    !***********************************************************
    !
    ! Procedure main
    !
    !   This is the entry point of your program
    !
    !***********************************************************
    PROC main()
        Path_10;
      !Add your code here
    ENDPROC
      PROC Path_10()
SetDO drillDone,0;
MoveAbsJ jHome, v100, fine, tool0\WObj:= wobj0;
WaitTime 2;
confL \Off;
confJ \Off;
        MoveJ RelTool(Target_10,0,0,-10),v60,z10,DrillTool\WObj:=FakeWing;
SetDO drillDone,1;
WaitUntil drillDone = 0;
        MoveL Target_10,v30,fine,DrillTool\WObj:=FakeWing;
SetDO drillDone,1;
WaitUntil drillDone = 0;
        MoveL RelTool(Target_10,0,0,-10),v30,z10,DrillTool\WObj:=FakeWing;
        MoveL RelTool(Target_20,0,0,-10),v30,z10,DrillTool\WObj:=FakeWing;
        MoveL Target_20,v30,fine,DrillTool\WObj:=FakeWing;
SetDO drillDone,1;
WaitUntil drillDone = 0;
        MoveL RelTool(Target_20,0,0,-10),v30,z10,DrillTool\WObj:=FakeWing;
        MoveL RelTool(Target_30,0,0,-10),v30,z10,DrillTool\WObj:=FakeWing;
        MoveL Target_30,v30,fine,DrillTool\WObj:=FakeWing;
SetDO drillDone,1;
WaitUntil drillDone = 0;
        MoveL RelTool(Target_30,0,0,-10),v30,z10,DrillTool\WObj:=FakeWing;
        MoveL RelTool(Target_40,0,0,-10),v30,z10,DrillTool\WObj:=FakeWing;
        MoveL Target_40,v30,fine,DrillTool\WObj:=FakeWing;
SetDO drillDone,1;
WaitUntil drillDone = 0;
        MoveL RelTool(Target_40,0,0,-10),v30,z10,DrillTool\WObj:=FakeWing;
        MoveL RelTool(Target_50,0,0,-10),v30,z10,DrillTool\WObj:=FakeWing;
        MoveL Target_50,v30,fine,DrillTool\WObj:=FakeWing;
SetDO drillDone,1;
WaitUntil drillDone = 0;
        MoveL RelTool(Target_50,0,0,-10),v30,z10,DrillTool\WObj:=FakeWing;
        MoveL RelTool(Target_60,0,0,-10),v30,z10,DrillTool\WObj:=FakeWing;
        MoveL Target_60,v30,fine,DrillTool\WObj:=FakeWing;
SetDO drillDone,1;
WaitUntil drillDone = 0;
        MoveL RelTool(Target_60,0,0,-10),v30,z10,DrillTool\WObj:=FakeWing;
        MoveL RelTool(Target_70,0,0,-10),v30,z10,DrillTool\WObj:=FakeWing;
        MoveL Target_70,v30,fine,DrillTool\WObj:=FakeWing;
SetDO drillDone,1;
WaitUntil drillDone = 0;
        MoveL RelTool(Target_70,0,0,-10),v30,z10,DrillTool\WObj:=FakeWing;
        MoveL RelTool(Target_80,0,0,-10),v30,z10,DrillTool\WObj:=FakeWing;
        MoveL Target_80,v30,fine,DrillTool\WObj:=FakeWing;
SetDO drillDone,1;
WaitUntil drillDone = 0;
        MoveL RelTool(Target_80,0,0,-10),v30,z10,DrillTool\WObj:=FakeWing;
        MoveL RelTool(Target_90,0,0,-10),v30,z10,DrillTool\WObj:=FakeWing;
        MoveL Target_90,v30,fine,DrillTool\WObj:=FakeWing;
SetDO drillDone,1;
WaitUntil drillDone = 0;
        MoveL RelTool(Target_90,0,0,-10),v30,z10,DrillTool\WObj:=FakeWing;
        MoveL RelTool(Target_100,0,0,-10),v30,z10,DrillTool\WObj:=FakeWing;
        MoveL Target_100,v30,fine,DrillTool\WObj:=FakeWing;
SetDO drillDone,1;
WaitUntil drillDone = 0;
        MoveL RelTool(Target_100,0,0,-10),v30,z10,DrillTool\WObj:=FakeWing;
        MoveL RelTool(Target_110,0,0,-10),v30,z10,DrillTool\WObj:=FakeWing;
        MoveL Target_110,v30,fine,DrillTool\WObj:=FakeWing;
SetDO drillDone,1;
WaitUntil drillDone = 0;
        MoveL RelTool(Target_110,0,0,-10),v30,z10,DrillTool\WObj:=FakeWing;
        MoveL RelTool(Target_120,0,0,-10),v30,z10,DrillTool\WObj:=FakeWing;
        MoveL Target_120,v30,fine,DrillTool\WObj:=FakeWing;
SetDO drillDone,1;
WaitUntil drillDone = 0;
        MoveL RelTool(Target_120,0,0,-10),v30,z10,DrillTool\WObj:=FakeWing;
        MoveL RelTool(Target_130,0,0,-10),v30,z10,DrillTool\WObj:=FakeWing;
        MoveL Target_130,v30,fine,DrillTool\WObj:=FakeWing;
SetDO drillDone,1;
WaitUntil drillDone = 0;
        MoveL RelTool(Target_130,0,0,-10),v30,z10,DrillTool\WObj:=FakeWing;
        MoveL RelTool(Target_140,0,0,-10),v30,z10,DrillTool\WObj:=FakeWing;
        MoveL Target_140,v30,fine,DrillTool\WObj:=FakeWing;
SetDO drillDone,1;
WaitUntil drillDone = 0;
        MoveL RelTool(Target_140,0,0,-10),v30,z10,DrillTool\WObj:=FakeWing;
        MoveL RelTool(Target_150,0,0,-10),v30,z10,DrillTool\WObj:=FakeWing;
        MoveL Target_150,v30,fine,DrillTool\WObj:=FakeWing;
SetDO drillDone,1;
WaitUntil drillDone = 0;
        MoveL RelTool(Target_150,0,0,-10),v30,z10,DrillTool\WObj:=FakeWing;
        MoveL RelTool(Target_160,0,0,-10),v30,z10,DrillTool\WObj:=FakeWing;
        MoveL Target_160,v30,fine,DrillTool\WObj:=FakeWing;
SetDO drillDone,1;
WaitUntil drillDone = 0;
        MoveL RelTool(Target_160,0,0,-10),v30,z10,DrillTool\WObj:=FakeWing;
        MoveL RelTool(Target_170,0,0,-10),v30,z10,DrillTool\WObj:=FakeWing;
        MoveL Target_170,v30,fine,DrillTool\WObj:=FakeWing;
SetDO drillDone,1;
WaitUntil drillDone = 0;
        MoveL RelTool(Target_170,0,0,-10),v30,z10,DrillTool\WObj:=FakeWing;
        MoveL RelTool(Target_180,0,0,-10),v30,z10,DrillTool\WObj:=FakeWing;
        MoveL Target_180,v30,fine,DrillTool\WObj:=FakeWing;
SetDO drillDone,1;
WaitUntil drillDone = 0;
        MoveL RelTool(Target_180,0,0,-10),v30,z10,DrillTool\WObj:=FakeWing;
        MoveL RelTool(Target_190,0,0,-10),v30,z10,DrillTool\WObj:=FakeWing;
        MoveL Target_190,v30,fine,DrillTool\WObj:=FakeWing;
SetDO drillDone,1;
WaitUntil drillDone = 0;
        MoveL RelTool(Target_190,0,0,-10),v30,z10,DrillTool\WObj:=FakeWing;
        MoveL RelTool(Target_200,0,0,-10),v30,z10,DrillTool\WObj:=FakeWing;
        MoveL Target_200,v30,fine,DrillTool\WObj:=FakeWing;
SetDO drillDone,1;
WaitUntil drillDone = 0;
        MoveL RelTool(Target_200,0,0,-10),v30,z10,DrillTool\WObj:=FakeWing;
        MoveL RelTool(Target_210,0,0,-10),v30,z10,DrillTool\WObj:=FakeWing;
        MoveL Target_210,v30,fine,DrillTool\WObj:=FakeWing;
SetDO drillDone,1;
WaitUntil drillDone = 0;
        MoveL RelTool(Target_210,0,0,-10),v30,z10,DrillTool\WObj:=FakeWing;
        MoveL RelTool(Target_220,0,0,-10),v30,z10,DrillTool\WObj:=FakeWing;
        MoveL Target_220,v30,fine,DrillTool\WObj:=FakeWing;
SetDO drillDone,1;
WaitUntil drillDone = 0;
        MoveL RelTool(Target_220,0,0,-10),v30,z10,DrillTool\WObj:=FakeWing;
        MoveL RelTool(Target_230,0,0,-10),v30,z10,DrillTool\WObj:=FakeWing;
        MoveL Target_230,v30,fine,DrillTool\WObj:=FakeWing;
SetDO drillDone,1;
WaitUntil drillDone = 0;
        MoveL RelTool(Target_230,0,0,-10),v30,z10,DrillTool\WObj:=FakeWing;
        MoveL RelTool(Target_240,0,0,-10),v30,z10,DrillTool\WObj:=FakeWing;
        MoveL Target_240,v30,fine,DrillTool\WObj:=FakeWing;
SetDO drillDone,1;
WaitUntil drillDone = 0;
        MoveL RelTool(Target_240,0,0,-10),v30,z10,DrillTool\WObj:=FakeWing;
        MoveL RelTool(Target_250,0,0,-10),v30,z10,DrillTool\WObj:=FakeWing;
        MoveL Target_250,v30,fine,DrillTool\WObj:=FakeWing;
SetDO drillDone,1;
WaitUntil drillDone = 0;
        MoveL RelTool(Target_250,0,0,-10),v30,z10,DrillTool\WObj:=FakeWing;
        MoveL RelTool(Target_260,0,0,-10),v30,z10,DrillTool\WObj:=FakeWing;
        MoveL Target_260,v30,fine,DrillTool\WObj:=FakeWing;
SetDO drillDone,1;
WaitUntil drillDone = 0;
        MoveL RelTool(Target_260,0,0,-10),v30,z10,DrillTool\WObj:=FakeWing;
        MoveL RelTool(Target_270,0,0,-10),v30,z10,DrillTool\WObj:=FakeWing;
        MoveL Target_270,v30,fine,DrillTool\WObj:=FakeWing;
SetDO drillDone,1;
WaitUntil drillDone = 0;
        MoveL RelTool(Target_270,0,0,-10),v30,z10,DrillTool\WObj:=FakeWing;
        MoveL RelTool(Target_280,0,0,-10),v30,z10,DrillTool\WObj:=FakeWing;
        MoveL Target_280,v30,fine,DrillTool\WObj:=FakeWing;
SetDO drillDone,1;
WaitUntil drillDone = 0;
        MoveL RelTool(Target_280,0,0,-10),v30,z10,DrillTool\WObj:=FakeWing;
        MoveL RelTool(Target_290,0,0,-10),v30,z10,DrillTool\WObj:=FakeWing;
        MoveL Target_290,v30,fine,DrillTool\WObj:=FakeWing;
SetDO drillDone,1;
WaitUntil drillDone = 0;
        MoveL RelTool(Target_290,0,0,-10),v30,z10,DrillTool\WObj:=FakeWing;
        MoveL RelTool(Target_300,0,0,-10),v30,z10,DrillTool\WObj:=FakeWing;
        MoveL Target_300,v30,fine,DrillTool\WObj:=FakeWing;
SetDO drillDone,1;
WaitUntil drillDone = 0;
        MoveL RelTool(Target_300,0,0,-10),v30,z10,DrillTool\WObj:=FakeWing;
        MoveL RelTool(Target_310,0,0,-10),v30,z10,DrillTool\WObj:=FakeWing;
        MoveL Target_310,v30,fine,DrillTool\WObj:=FakeWing;
SetDO drillDone,1;
WaitUntil drillDone = 0;
        MoveL RelTool(Target_310,0,0,-10),v30,z10,DrillTool\WObj:=FakeWing;
        MoveL RelTool(Target_320,0,0,-10),v30,z10,DrillTool\WObj:=FakeWing;
        MoveL Target_320,v30,fine,DrillTool\WObj:=FakeWing;
SetDO drillDone,1;
WaitUntil drillDone = 0;
        MoveL RelTool(Target_320,0,0,-10),v30,z10,DrillTool\WObj:=FakeWing;
        MoveL RelTool(Target_330,0,0,-10),v30,z10,DrillTool\WObj:=FakeWing;
        MoveL Target_330,v30,fine,DrillTool\WObj:=FakeWing;
SetDO drillDone,1;
WaitUntil drillDone = 0;
        MoveL RelTool(Target_330,0,0,-10),v30,z10,DrillTool\WObj:=FakeWing;
        MoveL RelTool(Target_340,0,0,-10),v30,z10,DrillTool\WObj:=FakeWing;
        MoveL Target_340,v30,fine,DrillTool\WObj:=FakeWing;
SetDO drillDone,1;
WaitUntil drillDone = 0;
        MoveL RelTool(Target_340,0,0,-10),v30,z10,DrillTool\WObj:=FakeWing;
        MoveL RelTool(Target_350,0,0,-10),v30,z10,DrillTool\WObj:=FakeWing;
        MoveL Target_350,v30,fine,DrillTool\WObj:=FakeWing;
SetDO drillDone,1;
WaitUntil drillDone = 0;
        MoveL RelTool(Target_350,0,0,-10),v30,z10,DrillTool\WObj:=FakeWing;
        MoveL RelTool(Target_360,0,0,-10),v30,z10,DrillTool\WObj:=FakeWing;
        MoveL Target_360,v30,fine,DrillTool\WObj:=FakeWing;
SetDO drillDone,1;
WaitUntil drillDone = 0;
        MoveL RelTool(Target_360,0,0,-10),v30,z10,DrillTool\WObj:=FakeWing;
        MoveL RelTool(Target_370,0,0,-10),v30,z10,DrillTool\WObj:=FakeWing;
        MoveL Target_370,v30,fine,DrillTool\WObj:=FakeWing;
SetDO drillDone,1;
WaitUntil drillDone = 0;
        MoveL RelTool(Target_370,0,0,-10),v30,z10,DrillTool\WObj:=FakeWing;
        MoveL RelTool(Target_380,0,0,-10),v30,z10,DrillTool\WObj:=FakeWing;
        MoveL Target_380,v30,fine,DrillTool\WObj:=FakeWing;
SetDO drillDone,1;
WaitUntil drillDone = 0;
        MoveL RelTool(Target_380,0,0,-10),v30,z10,DrillTool\WObj:=FakeWing;
        MoveL RelTool(Target_390,0,0,-10),v30,z10,DrillTool\WObj:=FakeWing;
        MoveL Target_390,v30,fine,DrillTool\WObj:=FakeWing;
SetDO drillDone,1;
WaitUntil drillDone = 0;
        MoveL RelTool(Target_390,0,0,-10),v30,z10,DrillTool\WObj:=FakeWing;
        MoveL RelTool(Target_400,0,0,-10),v30,z10,DrillTool\WObj:=FakeWing;
        MoveL Target_400,v30,fine,DrillTool\WObj:=FakeWing;
SetDO drillDone,1;
WaitUntil drillDone = 0;
        MoveL RelTool(Target_400,0,0,-10),v30,z10,DrillTool\WObj:=FakeWing;
        MoveL RelTool(Target_410,0,0,-10),v30,z10,DrillTool\WObj:=FakeWing;
        MoveL Target_410,v30,fine,DrillTool\WObj:=FakeWing;
SetDO drillDone,1;
WaitUntil drillDone = 0;
        MoveL RelTool(Target_410,0,0,-10),v30,z10,DrillTool\WObj:=FakeWing;
        MoveL RelTool(Target_420,0,0,-10),v30,z10,DrillTool\WObj:=FakeWing;
        MoveL Target_420,v30,fine,DrillTool\WObj:=FakeWing;
SetDO drillDone,1;
WaitUntil drillDone = 0;
        MoveL RelTool(Target_420,0,0,-10),v30,z10,DrillTool\WObj:=FakeWing;
        MoveL RelTool(Target_430,0,0,-10),v30,z10,DrillTool\WObj:=FakeWing;
        MoveL Target_430,v30,fine,DrillTool\WObj:=FakeWing;
SetDO drillDone,1;
WaitUntil drillDone = 0;
        MoveL RelTool(Target_430,0,0,-10),v30,z10,DrillTool\WObj:=FakeWing;
        MoveL RelTool(Target_440,0,0,-10),v30,z10,DrillTool\WObj:=FakeWing;
        MoveL Target_440,v30,fine,DrillTool\WObj:=FakeWing;
SetDO drillDone,1;
WaitUntil drillDone = 0;
        MoveL RelTool(Target_440,0,0,-10),v30,z10,DrillTool\WObj:=FakeWing;
        MoveL RelTool(Target_450,0,0,-10),v30,z10,DrillTool\WObj:=FakeWing;
        MoveL Target_450,v30,fine,DrillTool\WObj:=FakeWing;
SetDO drillDone,1;
WaitUntil drillDone = 0;
        MoveL RelTool(Target_450,0,0,-10),v30,z10,DrillTool\WObj:=FakeWing;
        MoveL RelTool(Target_460,0,0,-10),v30,z10,DrillTool\WObj:=FakeWing;
        MoveL Target_460,v30,fine,DrillTool\WObj:=FakeWing;
SetDO drillDone,1;
WaitUntil drillDone = 0;
        MoveL RelTool(Target_460,0,0,-10),v30,z10,DrillTool\WObj:=FakeWing;
        MoveL RelTool(Target_470,0,0,-10),v30,z10,DrillTool\WObj:=FakeWing;
        MoveL Target_470,v30,fine,DrillTool\WObj:=FakeWing;
SetDO drillDone,1;
WaitUntil drillDone = 0;
        MoveL RelTool(Target_470,0,0,-10),v30,z10,DrillTool\WObj:=FakeWing;
        MoveL RelTool(Target_480,0,0,-10),v30,z10,DrillTool\WObj:=FakeWing;
        MoveL Target_480,v30,fine,DrillTool\WObj:=FakeWing;
SetDO drillDone,1;
WaitUntil drillDone = 0;
        MoveL RelTool(Target_480,0,0,-10),v30,z10,DrillTool\WObj:=FakeWing;
        MoveL RelTool(Target_490,0,0,-10),v30,z10,DrillTool\WObj:=FakeWing;
        MoveL Target_490,v30,fine,DrillTool\WObj:=FakeWing;
SetDO drillDone,1;
WaitUntil drillDone = 0;
        MoveL RelTool(Target_490,0,0,-10),v30,z10,DrillTool\WObj:=FakeWing;
        MoveL RelTool(Target_500,0,0,-10),v30,z10,DrillTool\WObj:=FakeWing;
        MoveL Target_500,v30,fine,DrillTool\WObj:=FakeWing;
SetDO drillDone,1;
WaitUntil drillDone = 0;
        MoveL RelTool(Target_500,0,0,-10),v30,z10,DrillTool\WObj:=FakeWing;
        MoveL RelTool(Target_510,0,0,-10),v30,z10,DrillTool\WObj:=FakeWing;
        MoveL Target_510,v30,fine,DrillTool\WObj:=FakeWing;
SetDO drillDone,1;
WaitUntil drillDone = 0;
        MoveL RelTool(Target_510,0,0,-10),v30,z10,DrillTool\WObj:=FakeWing;
        MoveL RelTool(Target_520,0,0,-10),v30,z10,DrillTool\WObj:=FakeWing;
        MoveL Target_520,v30,fine,DrillTool\WObj:=FakeWing;
SetDO drillDone,1;
WaitUntil drillDone = 0;
        MoveL RelTool(Target_520,0,0,-10),v30,z10,DrillTool\WObj:=FakeWing;
        MoveL RelTool(Target_530,0,0,-10),v30,z10,DrillTool\WObj:=FakeWing;
        MoveL Target_530,v30,fine,DrillTool\WObj:=FakeWing;
SetDO drillDone,1;
WaitUntil drillDone = 0;
        MoveL RelTool(Target_530,0,0,-10),v30,z10,DrillTool\WObj:=FakeWing;
        MoveL RelTool(Target_540,0,0,-10),v30,z10,DrillTool\WObj:=FakeWing;
        MoveL Target_540,v30,fine,DrillTool\WObj:=FakeWing;
SetDO drillDone,1;
WaitUntil drillDone = 0;
        MoveL RelTool(Target_540,0,0,-10),v30,z10,DrillTool\WObj:=FakeWing;
        MoveL RelTool(Target_550,0,0,-10),v30,z10,DrillTool\WObj:=FakeWing;
        MoveL Target_550,v30,fine,DrillTool\WObj:=FakeWing;
SetDO drillDone,1;
WaitUntil drillDone = 0;
        MoveL RelTool(Target_550,0,0,-10),v30,z10,DrillTool\WObj:=FakeWing;
        MoveL RelTool(Target_560,0,0,-10),v30,z10,DrillTool\WObj:=FakeWing;
        MoveL Target_560,v30,fine,DrillTool\WObj:=FakeWing;
SetDO drillDone,1;
WaitUntil drillDone = 0;
        MoveL RelTool(Target_560,0,0,-10),v30,z10,DrillTool\WObj:=FakeWing;
        MoveL RelTool(Target_570,0,0,-10),v30,z10,DrillTool\WObj:=FakeWing;
        MoveL Target_570,v30,fine,DrillTool\WObj:=FakeWing;
SetDO drillDone,1;
WaitUntil drillDone = 0;
        MoveL RelTool(Target_570,0,0,-10),v30,z10,DrillTool\WObj:=FakeWing;
        MoveL RelTool(Target_580,0,0,-10),v30,z10,DrillTool\WObj:=FakeWing;
        MoveL Target_580,v30,fine,DrillTool\WObj:=FakeWing;
SetDO drillDone,1;
WaitUntil drillDone = 0;
        MoveL RelTool(Target_580,0,0,-10),v30,z10,DrillTool\WObj:=FakeWing;
        MoveL RelTool(Target_590,0,0,-10),v30,z10,DrillTool\WObj:=FakeWing;
        MoveL Target_590,v30,fine,DrillTool\WObj:=FakeWing;
SetDO drillDone,1;
WaitUntil drillDone = 0;
        MoveL RelTool(Target_590,0,0,-10),v30,z10,DrillTool\WObj:=FakeWing;
        MoveL RelTool(Target_600,0,0,-10),v30,z10,DrillTool\WObj:=FakeWing;
        MoveL Target_600,v30,fine,DrillTool\WObj:=FakeWing;
SetDO drillDone,1;
WaitUntil drillDone = 0;
        MoveL RelTool(Target_600,0,0,-10),v30,z10,DrillTool\WObj:=FakeWing;
        MoveL RelTool(Target_610,0,0,-10),v30,z10,DrillTool\WObj:=FakeWing;
        MoveL Target_610,v30,fine,DrillTool\WObj:=FakeWing;
SetDO drillDone,1;
WaitUntil drillDone = 0;
        MoveL RelTool(Target_610,0,0,-10),v30,z10,DrillTool\WObj:=FakeWing;
        MoveL RelTool(Target_620,0,0,-10),v30,z10,DrillTool\WObj:=FakeWing;
        MoveL Target_620,v30,fine,DrillTool\WObj:=FakeWing;
SetDO drillDone,1;
WaitUntil drillDone = 0;
        MoveL RelTool(Target_620,0,0,-10),v30,z10,DrillTool\WObj:=FakeWing;
        MoveL RelTool(Target_630,0,0,-10),v30,z10,DrillTool\WObj:=FakeWing;
        MoveL Target_630,v30,fine,DrillTool\WObj:=FakeWing;
SetDO drillDone,1;
WaitUntil drillDone = 0;
        MoveL RelTool(Target_630,0,0,-10),v30,z10,DrillTool\WObj:=FakeWing;
        MoveL RelTool(Target_640,0,0,-10),v30,z10,DrillTool\WObj:=FakeWing;
        MoveL Target_640,v30,fine,DrillTool\WObj:=FakeWing;
SetDO drillDone,1;
WaitUntil drillDone = 0;
        MoveL RelTool(Target_640,0,0,-10),v30,z10,DrillTool\WObj:=FakeWing;
        MoveL RelTool(Target_650,0,0,-10),v30,z10,DrillTool\WObj:=FakeWing;
        MoveL Target_650,v30,fine,DrillTool\WObj:=FakeWing;
SetDO drillDone,1;
WaitUntil drillDone = 0;
        MoveL RelTool(Target_650,0,0,-10),v30,z10,DrillTool\WObj:=FakeWing;
        MoveL RelTool(Target_660,0,0,-10),v30,z10,DrillTool\WObj:=FakeWing;
        MoveL Target_660,v30,fine,DrillTool\WObj:=FakeWing;
SetDO drillDone,1;
WaitUntil drillDone = 0;
        MoveL RelTool(Target_660,0,0,-10),v30,z10,DrillTool\WObj:=FakeWing;
        MoveL RelTool(Target_670,0,0,-10),v30,z10,DrillTool\WObj:=FakeWing;
        MoveL Target_670,v30,fine,DrillTool\WObj:=FakeWing;
SetDO drillDone,1;
WaitUntil drillDone = 0;
        MoveL RelTool(Target_670,0,0,-10),v30,z10,DrillTool\WObj:=FakeWing;
        MoveL RelTool(Target_680,0,0,-10),v30,z10,DrillTool\WObj:=FakeWing;
        MoveL Target_680,v30,fine,DrillTool\WObj:=FakeWing;
SetDO drillDone,1;
WaitUntil drillDone = 0;
        MoveL RelTool(Target_680,0,0,-10),v30,z10,DrillTool\WObj:=FakeWing;
        MoveL RelTool(Target_690,0,0,-10),v30,z10,DrillTool\WObj:=FakeWing;
        MoveL Target_690,v30,fine,DrillTool\WObj:=FakeWing;
SetDO drillDone,1;
WaitUntil drillDone = 0;
        MoveL RelTool(Target_690,0,0,-10),v30,z10,DrillTool\WObj:=FakeWing;
        MoveL RelTool(Target_700,0,0,-10),v30,z10,DrillTool\WObj:=FakeWing;
        MoveL Target_700,v30,fine,DrillTool\WObj:=FakeWing;
SetDO drillDone,1;
WaitUntil drillDone = 0;
        MoveL RelTool(Target_700,0,0,-10),v30,z10,DrillTool\WObj:=FakeWing;
        MoveL RelTool(Target_710,0,0,-10),v30,z10,DrillTool\WObj:=FakeWing;
        MoveL Target_710,v30,fine,DrillTool\WObj:=FakeWing;
SetDO drillDone,1;
WaitUntil drillDone = 0;
        MoveL RelTool(Target_710,0,0,-10),v30,z10,DrillTool\WObj:=FakeWing;
        MoveL RelTool(Target_720,0,0,-10),v30,z10,DrillTool\WObj:=FakeWing;
        MoveL Target_720,v30,fine,DrillTool\WObj:=FakeWing;
SetDO drillDone,1;
WaitUntil drillDone = 0;
        MoveL RelTool(Target_720,0,0,-10),v30,z10,DrillTool\WObj:=FakeWing;
        MoveL RelTool(Target_730,0,0,-10),v30,z10,DrillTool\WObj:=FakeWing;
        MoveL Target_730,v30,fine,DrillTool\WObj:=FakeWing;
SetDO drillDone,1;
WaitUntil drillDone = 0;
        MoveL RelTool(Target_730,0,0,-10),v30,z10,DrillTool\WObj:=FakeWing;
        MoveL RelTool(Target_740,0,0,-10),v30,z10,DrillTool\WObj:=FakeWing;
        MoveL Target_740,v30,fine,DrillTool\WObj:=FakeWing;
SetDO drillDone,1;
WaitUntil drillDone = 0;
        MoveL RelTool(Target_740,0,0,-10),v30,z10,DrillTool\WObj:=FakeWing;
        MoveL RelTool(Target_750,0,0,-10),v30,z10,DrillTool\WObj:=FakeWing;
        MoveL Target_750,v30,fine,DrillTool\WObj:=FakeWing;
SetDO drillDone,1;
WaitUntil drillDone = 0;
        MoveL RelTool(Target_750,0,0,-10),v30,z10,DrillTool\WObj:=FakeWing;
        MoveL RelTool(Target_760,0,0,-10),v30,z10,DrillTool\WObj:=FakeWing;
        MoveL Target_760,v30,fine,DrillTool\WObj:=FakeWing;
SetDO drillDone,1;
WaitUntil drillDone = 0;
        MoveL RelTool(Target_760,0,0,-10),v30,z10,DrillTool\WObj:=FakeWing;
        MoveL RelTool(Target_770,0,0,-10),v30,z10,DrillTool\WObj:=FakeWing;
        MoveL Target_770,v30,fine,DrillTool\WObj:=FakeWing;
SetDO drillDone,1;
WaitUntil drillDone = 0;
        MoveL RelTool(Target_770,0,0,-10),v30,z10,DrillTool\WObj:=FakeWing;
        MoveL RelTool(Target_780,0,0,-10),v30,z10,DrillTool\WObj:=FakeWing;
        MoveL Target_780,v30,fine,DrillTool\WObj:=FakeWing;
SetDO drillDone,1;
WaitUntil drillDone = 0;
        MoveL RelTool(Target_780,0,0,-10),v30,z10,DrillTool\WObj:=FakeWing;
        MoveL RelTool(Target_790,0,0,-10),v30,z10,DrillTool\WObj:=FakeWing;
        MoveL Target_790,v30,fine,DrillTool\WObj:=FakeWing;
SetDO drillDone,1;
WaitUntil drillDone = 0;
        MoveL RelTool(Target_790,0,0,-10),v30,z10,DrillTool\WObj:=FakeWing;
        MoveL RelTool(Target_800,0,0,-10),v30,z10,DrillTool\WObj:=FakeWing;
        MoveL Target_800,v30,fine,DrillTool\WObj:=FakeWing;
SetDO drillDone,1;
WaitUntil drillDone = 0;
        MoveL RelTool(Target_800,0,0,-10),v30,z10,DrillTool\WObj:=FakeWing;
        MoveL RelTool(Target_810,0,0,-10),v30,z10,DrillTool\WObj:=FakeWing;
        MoveL Target_810,v30,fine,DrillTool\WObj:=FakeWing;
SetDO drillDone,1;
WaitUntil drillDone = 0;
        MoveL RelTool(Target_810,0,0,-10),v30,z10,DrillTool\WObj:=FakeWing;
        MoveL RelTool(Target_820,0,0,-10),v30,z10,DrillTool\WObj:=FakeWing;
        MoveL Target_820,v30,fine,DrillTool\WObj:=FakeWing;
SetDO drillDone,1;
WaitUntil drillDone = 0;
        MoveL RelTool(Target_820,0,0,-10),v30,z10,DrillTool\WObj:=FakeWing;
        MoveL RelTool(Target_830,0,0,-10),v30,z10,DrillTool\WObj:=FakeWing;
        MoveL Target_830,v30,fine,DrillTool\WObj:=FakeWing;
SetDO drillDone,1;
WaitUntil drillDone = 0;
        MoveL RelTool(Target_830,0,0,-10),v30,z10,DrillTool\WObj:=FakeWing;
        MoveL RelTool(Target_840,0,0,-10),v30,z10,DrillTool\WObj:=FakeWing;
        MoveL Target_840,v30,fine,DrillTool\WObj:=FakeWing;
SetDO drillDone,1;
WaitUntil drillDone = 0;
        MoveL RelTool(Target_840,0,0,-10),v30,z10,DrillTool\WObj:=FakeWing;
        MoveL RelTool(Target_850,0,0,-10),v30,z10,DrillTool\WObj:=FakeWing;
        MoveL Target_850,v30,fine,DrillTool\WObj:=FakeWing;
SetDO drillDone,1;
WaitUntil drillDone = 0;
        MoveL RelTool(Target_850,0,0,-10),v30,z10,DrillTool\WObj:=FakeWing;
        MoveL RelTool(Target_860,0,0,-10),v30,z10,DrillTool\WObj:=FakeWing;
        MoveL Target_860,v30,fine,DrillTool\WObj:=FakeWing;
SetDO drillDone,1;
WaitUntil drillDone = 0;
        MoveL RelTool(Target_860,0,0,-10),v30,z10,DrillTool\WObj:=FakeWing;
        MoveL RelTool(Target_870,0,0,-10),v30,z10,DrillTool\WObj:=FakeWing;
        MoveL Target_870,v30,fine,DrillTool\WObj:=FakeWing;
SetDO drillDone,1;
WaitUntil drillDone = 0;
        MoveL RelTool(Target_870,0,0,-10),v30,z10,DrillTool\WObj:=FakeWing;
        MoveL RelTool(Target_880,0,0,-10),v30,z10,DrillTool\WObj:=FakeWing;
        MoveL Target_880,v30,fine,DrillTool\WObj:=FakeWing;
SetDO drillDone,1;
WaitUntil drillDone = 0;
        MoveL RelTool(Target_880,0,0,-10),v30,z10,DrillTool\WObj:=FakeWing;
        MoveL RelTool(Target_890,0,0,-10),v30,z10,DrillTool\WObj:=FakeWing;
        MoveL Target_890,v30,fine,DrillTool\WObj:=FakeWing;
SetDO drillDone,1;
WaitUntil drillDone = 0;
        MoveL RelTool(Target_890,0,0,-10),v30,z10,DrillTool\WObj:=FakeWing;
        MoveL RelTool(Target_900,0,0,-10),v30,z10,DrillTool\WObj:=FakeWing;
        MoveL Target_900,v30,fine,DrillTool\WObj:=FakeWing;
SetDO drillDone,1;
WaitUntil drillDone = 0;
        MoveL RelTool(Target_900,0,0,-10),v30,z10,DrillTool\WObj:=FakeWing;
        MoveL RelTool(Target_910,0,0,-10),v30,z10,DrillTool\WObj:=FakeWing;
        MoveL Target_910,v30,fine,DrillTool\WObj:=FakeWing;
SetDO drillDone,1;
WaitUntil drillDone = 0;
        MoveL RelTool(Target_910,0,0,-10),v30,z10,DrillTool\WObj:=FakeWing;
        MoveL RelTool(Target_920,0,0,-10),v30,z10,DrillTool\WObj:=FakeWing;
        MoveL Target_920,v30,fine,DrillTool\WObj:=FakeWing;
SetDO drillDone,1;
WaitUntil drillDone = 0;
        MoveL RelTool(Target_920,0,0,-10),v30,z10,DrillTool\WObj:=FakeWing;
        MoveL RelTool(Target_930,0,0,-10),v30,z10,DrillTool\WObj:=FakeWing;
        MoveL Target_930,v30,fine,DrillTool\WObj:=FakeWing;
SetDO drillDone,1;
WaitUntil drillDone = 0;
        MoveL RelTool(Target_930,0,0,-10),v30,z10,DrillTool\WObj:=FakeWing;
        MoveL RelTool(Target_940,0,0,-10),v30,z10,DrillTool\WObj:=FakeWing;
        MoveL Target_940,v30,fine,DrillTool\WObj:=FakeWing;
SetDO drillDone,1;
WaitUntil drillDone = 0;
        MoveL RelTool(Target_940,0,0,-10),v30,z10,DrillTool\WObj:=FakeWing;
        MoveL RelTool(Target_950,0,0,-10),v30,z10,DrillTool\WObj:=FakeWing;
        MoveL Target_950,v30,fine,DrillTool\WObj:=FakeWing;
SetDO drillDone,1;
WaitUntil drillDone = 0;
        MoveL RelTool(Target_950,0,0,-10),v30,z10,DrillTool\WObj:=FakeWing;
        MoveL RelTool(Target_960,0,0,-10),v30,z10,DrillTool\WObj:=FakeWing;
        MoveL Target_960,v30,fine,DrillTool\WObj:=FakeWing;
SetDO drillDone,1;
WaitUntil drillDone = 0;
        MoveL RelTool(Target_960,0,0,-10),v30,z10,DrillTool\WObj:=FakeWing;
        MoveL RelTool(Target_970,0,0,-10),v30,z10,DrillTool\WObj:=FakeWing;
        MoveL Target_970,v30,fine,DrillTool\WObj:=FakeWing;
SetDO drillDone,1;
WaitUntil drillDone = 0;
        MoveL RelTool(Target_970,0,0,-10),v30,z10,DrillTool\WObj:=FakeWing;
        MoveL RelTool(Target_980,0,0,-10),v30,z10,DrillTool\WObj:=FakeWing;
        MoveL Target_980,v30,fine,DrillTool\WObj:=FakeWing;
SetDO drillDone,1;
WaitUntil drillDone = 0;
        MoveL RelTool(Target_980,0,0,-10),v30,z10,DrillTool\WObj:=FakeWing;
        MoveL RelTool(Target_990,0,0,-10),v30,z10,DrillTool\WObj:=FakeWing;
        MoveL Target_990,v30,fine,DrillTool\WObj:=FakeWing;
SetDO drillDone,1;
WaitUntil drillDone = 0;
        MoveL RelTool(Target_990,0,0,-10),v30,z10,DrillTool\WObj:=FakeWing;
        MoveL RelTool(Target_1000,0,0,-10),v30,z10,DrillTool\WObj:=FakeWing;
        MoveL Target_1000,v30,fine,DrillTool\WObj:=FakeWing;
SetDO drillDone,1;
WaitUntil drillDone = 0;
        MoveL RelTool(Target_1000,0,0,-10),v30,z10,DrillTool\WObj:=FakeWing;
        MoveL RelTool(Target_1010,0,0,-10),v30,z10,DrillTool\WObj:=FakeWing;
        MoveL Target_1010,v30,fine,DrillTool\WObj:=FakeWing;
SetDO drillDone,1;
WaitUntil drillDone = 0;
        MoveL RelTool(Target_1010,0,0,-10),v30,z10,DrillTool\WObj:=FakeWing;
        MoveL RelTool(Target_1020,0,0,-10),v30,z10,DrillTool\WObj:=FakeWing;
        MoveL Target_1020,v30,fine,DrillTool\WObj:=FakeWing;
SetDO drillDone,1;
WaitUntil drillDone = 0;
        MoveL RelTool(Target_1020,0,0,-10),v30,z10,DrillTool\WObj:=FakeWing;
        MoveL RelTool(Target_1030,0,0,-10),v30,z10,DrillTool\WObj:=FakeWing;
        MoveL Target_1030,v30,fine,DrillTool\WObj:=FakeWing;
SetDO drillDone,1;
WaitUntil drillDone = 0;
        MoveL RelTool(Target_1030,0,0,-10),v30,z10,DrillTool\WObj:=FakeWing;
        MoveL RelTool(Target_1040,0,0,-10),v30,z10,DrillTool\WObj:=FakeWing;
        MoveL Target_1040,v30,fine,DrillTool\WObj:=FakeWing;
SetDO drillDone,1;
WaitUntil drillDone = 0;
        MoveL RelTool(Target_1040,0,0,-10),v30,z10,DrillTool\WObj:=FakeWing;
        MoveL RelTool(Target_1050,0,0,-10),v30,z10,DrillTool\WObj:=FakeWing;
        MoveL Target_1050,v30,fine,DrillTool\WObj:=FakeWing;
SetDO drillDone,1;
WaitUntil drillDone = 0;
        MoveL RelTool(Target_1050,0,0,-10),v30,z10,DrillTool\WObj:=FakeWing;
        MoveL RelTool(Target_1060,0,0,-10),v30,z10,DrillTool\WObj:=FakeWing;
        MoveL Target_1060,v30,fine,DrillTool\WObj:=FakeWing;
SetDO drillDone,1;
WaitUntil drillDone = 0;
        MoveL RelTool(Target_1060,0,0,-10),v30,z10,DrillTool\WObj:=FakeWing;
        MoveL RelTool(Target_1070,0,0,-10),v30,z10,DrillTool\WObj:=FakeWing;
        MoveL Target_1070,v30,fine,DrillTool\WObj:=FakeWing;
SetDO drillDone,1;
WaitUntil drillDone = 0;
        MoveL RelTool(Target_1070,0,0,-10),v30,z10,DrillTool\WObj:=FakeWing;
        MoveL RelTool(Target_1080,0,0,-10),v30,z10,DrillTool\WObj:=FakeWing;
        MoveL Target_1080,v30,fine,DrillTool\WObj:=FakeWing;
SetDO drillDone,1;
WaitUntil drillDone = 0;
        MoveL RelTool(Target_1080,0,0,-10),v30,z10,DrillTool\WObj:=FakeWing;
        MoveL RelTool(Target_1090,0,0,-10),v30,z10,DrillTool\WObj:=FakeWing;
        MoveL Target_1090,v30,fine,DrillTool\WObj:=FakeWing;
SetDO drillDone,1;
WaitUntil drillDone = 0;
        MoveL RelTool(Target_1090,0,0,-10),v30,z10,DrillTool\WObj:=FakeWing;
        MoveL RelTool(Target_1100,0,0,-10),v30,z10,DrillTool\WObj:=FakeWing;
        MoveL Target_1100,v30,fine,DrillTool\WObj:=FakeWing;
SetDO drillDone,1;
WaitUntil drillDone = 0;
        MoveL RelTool(Target_1100,0,0,-10),v30,z10,DrillTool\WObj:=FakeWing;
        MoveL RelTool(Target_1110,0,0,-10),v30,z10,DrillTool\WObj:=FakeWing;
        MoveL Target_1110,v30,fine,DrillTool\WObj:=FakeWing;
SetDO drillDone,1;
WaitUntil drillDone = 0;
        MoveL RelTool(Target_1110,0,0,-10),v30,z10,DrillTool\WObj:=FakeWing;
        MoveL RelTool(Target_1120,0,0,-10),v30,z10,DrillTool\WObj:=FakeWing;
        MoveL Target_1120,v30,fine,DrillTool\WObj:=FakeWing;
SetDO drillDone,1;
WaitUntil drillDone = 0;
        MoveL RelTool(Target_1120,0,0,-10),v30,z10,DrillTool\WObj:=FakeWing;
        MoveL RelTool(Target_1130,0,0,-10),v30,z10,DrillTool\WObj:=FakeWing;
        MoveL Target_1130,v30,fine,DrillTool\WObj:=FakeWing;
SetDO drillDone,1;
WaitUntil drillDone = 0;
        MoveL RelTool(Target_1130,0,0,-10),v30,z10,DrillTool\WObj:=FakeWing;
        MoveL RelTool(Target_1140,0,0,-10),v30,z10,DrillTool\WObj:=FakeWing;
        MoveL Target_1140,v30,fine,DrillTool\WObj:=FakeWing;
SetDO drillDone,1;
WaitUntil drillDone = 0;
        MoveL RelTool(Target_1140,0,0,-10),v30,z10,DrillTool\WObj:=FakeWing;
        MoveL RelTool(Target_1150,0,0,-10),v30,z10,DrillTool\WObj:=FakeWing;
        MoveL Target_1150,v30,fine,DrillTool\WObj:=FakeWing;
SetDO drillDone,1;
WaitUntil drillDone = 0;
        MoveL RelTool(Target_1150,0,0,-10),v30,z10,DrillTool\WObj:=FakeWing;
        MoveL RelTool(Target_1160,0,0,-10),v30,z10,DrillTool\WObj:=FakeWing;
        MoveL Target_1160,v30,fine,DrillTool\WObj:=FakeWing;
SetDO drillDone,1;
WaitUntil drillDone = 0;
        MoveL RelTool(Target_1160,0,0,-10),v30,z10,DrillTool\WObj:=FakeWing;
        MoveL RelTool(Target_1170,0,0,-10),v30,z10,DrillTool\WObj:=FakeWing;
        MoveL Target_1170,v30,fine,DrillTool\WObj:=FakeWing;
SetDO drillDone,1;
WaitUntil drillDone = 0;
        MoveL RelTool(Target_1170,0,0,-10),v30,z10,DrillTool\WObj:=FakeWing;
        MoveL RelTool(Target_1180,0,0,-10),v30,z10,DrillTool\WObj:=FakeWing;
        MoveL Target_1180,v30,fine,DrillTool\WObj:=FakeWing;
SetDO drillDone,1;
WaitUntil drillDone = 0;
        MoveL RelTool(Target_1180,0,0,-10),v30,z10,DrillTool\WObj:=FakeWing;
        MoveL RelTool(Target_1190,0,0,-10),v30,z10,DrillTool\WObj:=FakeWing;
        MoveL Target_1190,v30,fine,DrillTool\WObj:=FakeWing;
SetDO drillDone,1;
WaitUntil drillDone = 0;
        MoveL RelTool(Target_1190,0,0,-10),v30,z10,DrillTool\WObj:=FakeWing;
        MoveL RelTool(Target_1200,0,0,-10),v30,z10,DrillTool\WObj:=FakeWing;
        MoveL Target_1200,v30,fine,DrillTool\WObj:=FakeWing;
SetDO drillDone,1;
WaitUntil drillDone = 0;
        MoveL RelTool(Target_1200,0,0,-10),v30,z10,DrillTool\WObj:=FakeWing;
        MoveL RelTool(Target_1210,0,0,-10),v30,z10,DrillTool\WObj:=FakeWing;
        MoveL Target_1210,v30,fine,DrillTool\WObj:=FakeWing;
SetDO drillDone,1;
WaitUntil drillDone = 0;
        MoveL RelTool(Target_1210,0,0,-10),v30,z10,DrillTool\WObj:=FakeWing;
        MoveL RelTool(Target_1220,0,0,-10),v30,z10,DrillTool\WObj:=FakeWing;
        MoveL Target_1220,v30,fine,DrillTool\WObj:=FakeWing;
SetDO drillDone,1;
WaitUntil drillDone = 0;
        MoveL RelTool(Target_1220,0,0,-10),v30,z10,DrillTool\WObj:=FakeWing;
        MoveL RelTool(Target_1230,0,0,-10),v30,z10,DrillTool\WObj:=FakeWing;
        MoveL Target_1230,v30,fine,DrillTool\WObj:=FakeWing;
SetDO drillDone,1;
WaitUntil drillDone = 0;
        MoveL RelTool(Target_1230,0,0,-10),v30,z10,DrillTool\WObj:=FakeWing;
        MoveL RelTool(Target_1240,0,0,-10),v30,z10,DrillTool\WObj:=FakeWing;
        MoveL Target_1240,v30,fine,DrillTool\WObj:=FakeWing;
SetDO drillDone,1;
WaitUntil drillDone = 0;
        MoveL RelTool(Target_1240,0,0,-10),v30,z10,DrillTool\WObj:=FakeWing;
        MoveL RelTool(Target_1250,0,0,-10),v30,z10,DrillTool\WObj:=FakeWing;
        MoveL Target_1250,v30,fine,DrillTool\WObj:=FakeWing;
SetDO drillDone,1;
WaitUntil drillDone = 0;
        MoveL RelTool(Target_1250,0,0,-10),v30,z10,DrillTool\WObj:=FakeWing;
        MoveL RelTool(Target_1260,0,0,-10),v30,z10,DrillTool\WObj:=FakeWing;
        MoveL Target_1260,v30,fine,DrillTool\WObj:=FakeWing;
SetDO drillDone,1;
WaitUntil drillDone = 0;
        MoveL RelTool(Target_1260,0,0,-10),v30,z10,DrillTool\WObj:=FakeWing;
        MoveL RelTool(Target_1270,0,0,-10),v30,z10,DrillTool\WObj:=FakeWing;
        MoveL Target_1270,v30,fine,DrillTool\WObj:=FakeWing;
SetDO drillDone,1;
WaitUntil drillDone = 0;
        MoveL RelTool(Target_1270,0,0,-10),v30,z10,DrillTool\WObj:=FakeWing;
        MoveL RelTool(Target_1280,0,0,-10),v30,z10,DrillTool\WObj:=FakeWing;
        MoveL Target_1280,v30,fine,DrillTool\WObj:=FakeWing;
SetDO drillDone,1;
WaitUntil drillDone = 0;
        MoveL RelTool(Target_1280,0,0,-10),v30,z10,DrillTool\WObj:=FakeWing;
        MoveL RelTool(Target_1290,0,0,-10),v30,z10,DrillTool\WObj:=FakeWing;
        MoveL Target_1290,v30,fine,DrillTool\WObj:=FakeWing;
SetDO drillDone,1;
WaitUntil drillDone = 0;
        MoveL RelTool(Target_1290,0,0,-10),v30,z10,DrillTool\WObj:=FakeWing;
        MoveL RelTool(Target_1300,0,0,-10),v30,z10,DrillTool\WObj:=FakeWing;
        MoveL Target_1300,v30,fine,DrillTool\WObj:=FakeWing;
SetDO drillDone,1;
WaitUntil drillDone = 0;
        MoveL RelTool(Target_1300,0,0,-10),v30,z10,DrillTool\WObj:=FakeWing;
        MoveL RelTool(Target_1310,0,0,-10),v30,z10,DrillTool\WObj:=FakeWing;
        MoveL Target_1310,v30,fine,DrillTool\WObj:=FakeWing;
SetDO drillDone,1;
WaitUntil drillDone = 0;
        MoveL RelTool(Target_1310,0,0,-10),v30,z10,DrillTool\WObj:=FakeWing;
        MoveL RelTool(Target_1320,0,0,-10),v30,z10,DrillTool\WObj:=FakeWing;
        MoveL Target_1320,v30,fine,DrillTool\WObj:=FakeWing;
SetDO drillDone,1;
WaitUntil drillDone = 0;
        MoveL RelTool(Target_1320,0,0,-10),v30,z10,DrillTool\WObj:=FakeWing;
        MoveL RelTool(Target_1330,0,0,-10),v30,z10,DrillTool\WObj:=FakeWing;
        MoveL Target_1330,v30,fine,DrillTool\WObj:=FakeWing;
SetDO drillDone,1;
WaitUntil drillDone = 0;
        MoveL RelTool(Target_1330,0,0,-10),v30,z10,DrillTool\WObj:=FakeWing;
        MoveL RelTool(Target_1340,0,0,-10),v30,z10,DrillTool\WObj:=FakeWing;
        MoveL Target_1340,v30,fine,DrillTool\WObj:=FakeWing;
SetDO drillDone,1;
WaitUntil drillDone = 0;
        MoveL RelTool(Target_1340,0,0,-10),v30,z10,DrillTool\WObj:=FakeWing;
        MoveL RelTool(Target_1350,0,0,-10),v30,z10,DrillTool\WObj:=FakeWing;
        MoveL Target_1350,v30,fine,DrillTool\WObj:=FakeWing;
SetDO drillDone,1;
WaitUntil drillDone = 0;
        MoveL RelTool(Target_1350,0,0,-10),v30,z10,DrillTool\WObj:=FakeWing;
        MoveL RelTool(Target_1360,0,0,-10),v30,z10,DrillTool\WObj:=FakeWing;
        MoveL Target_1360,v30,fine,DrillTool\WObj:=FakeWing;
SetDO drillDone,1;
WaitUntil drillDone = 0;
        MoveL RelTool(Target_1360,0,0,-10),v30,z10,DrillTool\WObj:=FakeWing;
        MoveL RelTool(Target_1370,0,0,-10),v30,z10,DrillTool\WObj:=FakeWing;
        MoveL Target_1370,v30,fine,DrillTool\WObj:=FakeWing;
SetDO drillDone,1;
WaitUntil drillDone = 0;
        MoveL RelTool(Target_1370,0,0,-10),v30,z10,DrillTool\WObj:=FakeWing;
        MoveL RelTool(Target_1380,0,0,-10),v30,z10,DrillTool\WObj:=FakeWing;
        MoveL Target_1380,v30,fine,DrillTool\WObj:=FakeWing;
SetDO drillDone,1;
WaitUntil drillDone = 0;
        MoveL RelTool(Target_1380,0,0,-10),v30,z10,DrillTool\WObj:=FakeWing;
        MoveL RelTool(Target_1390,0,0,-10),v30,z10,DrillTool\WObj:=FakeWing;
        MoveL Target_1390,v30,fine,DrillTool\WObj:=FakeWing;
SetDO drillDone,1;
WaitUntil drillDone = 0;
        MoveL RelTool(Target_1390,0,0,-10),v30,z10,DrillTool\WObj:=FakeWing;
        MoveL RelTool(Target_1400,0,0,-10),v30,z10,DrillTool\WObj:=FakeWing;
        MoveL Target_1400,v30,fine,DrillTool\WObj:=FakeWing;
SetDO drillDone,1;
WaitUntil drillDone = 0;
        MoveL RelTool(Target_1400,0,0,-10),v30,z10,DrillTool\WObj:=FakeWing;
        MoveL RelTool(Target_1410,0,0,-10),v30,z10,DrillTool\WObj:=FakeWing;
        MoveL Target_1410,v30,fine,DrillTool\WObj:=FakeWing;
SetDO drillDone,1;
WaitUntil drillDone = 0;
        MoveL RelTool(Target_1410,0,0,-10),v30,z10,DrillTool\WObj:=FakeWing;
        MoveL RelTool(Target_1420,0,0,-10),v30,z10,DrillTool\WObj:=FakeWing;
        MoveL Target_1420,v30,fine,DrillTool\WObj:=FakeWing;
SetDO drillDone,1;
WaitUntil drillDone = 0;
        MoveL RelTool(Target_1420,0,0,-10),v30,z10,DrillTool\WObj:=FakeWing;
        MoveL RelTool(Target_1430,0,0,-10),v30,z10,DrillTool\WObj:=FakeWing;
        MoveL Target_1430,v30,fine,DrillTool\WObj:=FakeWing;
SetDO drillDone,1;
WaitUntil drillDone = 0;
        MoveL RelTool(Target_1430,0,0,-10),v30,z10,DrillTool\WObj:=FakeWing;
        MoveL RelTool(Target_1440,0,0,-10),v30,z10,DrillTool\WObj:=FakeWing;
        MoveL Target_1440,v30,fine,DrillTool\WObj:=FakeWing;
SetDO drillDone,1;
WaitUntil drillDone = 0;
        MoveL RelTool(Target_1440,0,0,-10),v30,z10,DrillTool\WObj:=FakeWing;
        MoveL RelTool(Target_1450,0,0,-10),v30,z10,DrillTool\WObj:=FakeWing;
        MoveL Target_1450,v30,fine,DrillTool\WObj:=FakeWing;
SetDO drillDone,1;
WaitUntil drillDone = 0;
        MoveL RelTool(Target_1450,0,0,-10),v30,z10,DrillTool\WObj:=FakeWing;
        MoveL RelTool(Target_1460,0,0,-10),v30,z10,DrillTool\WObj:=FakeWing;
        MoveL Target_1460,v30,fine,DrillTool\WObj:=FakeWing;
SetDO drillDone,1;
WaitUntil drillDone = 0;
        MoveL RelTool(Target_1460,0,0,-10),v30,z10,DrillTool\WObj:=FakeWing;
        MoveL RelTool(Target_1470,0,0,-10),v30,z10,DrillTool\WObj:=FakeWing;
        MoveL Target_1470,v30,fine,DrillTool\WObj:=FakeWing;
SetDO drillDone,1;
WaitUntil drillDone = 0;
        MoveL RelTool(Target_1470,0,0,-10),v30,z10,DrillTool\WObj:=FakeWing;
        MoveL RelTool(Target_1480,0,0,-10),v30,z10,DrillTool\WObj:=FakeWing;
        MoveL Target_1480,v30,fine,DrillTool\WObj:=FakeWing;
SetDO drillDone,1;
WaitUntil drillDone = 0;
        MoveL RelTool(Target_1480,0,0,-10),v30,z10,DrillTool\WObj:=FakeWing;
        MoveL RelTool(Target_1490,0,0,-10),v30,z10,DrillTool\WObj:=FakeWing;
        MoveL Target_1490,v30,fine,DrillTool\WObj:=FakeWing;
SetDO drillDone,1;
WaitUntil drillDone = 0;
        MoveL RelTool(Target_1490,0,0,-10),v30,z10,DrillTool\WObj:=FakeWing;
        MoveL RelTool(Target_1500,0,0,-10),v30,z10,DrillTool\WObj:=FakeWing;
        MoveL Target_1500,v30,fine,DrillTool\WObj:=FakeWing;
SetDO drillDone,1;
WaitUntil drillDone = 0;
        MoveL RelTool(Target_1500,0,0,-10),v30,z10,DrillTool\WObj:=FakeWing;
        MoveL RelTool(Target_1510,0,0,-10),v30,z10,DrillTool\WObj:=FakeWing;
        MoveL Target_1510,v30,fine,DrillTool\WObj:=FakeWing;
SetDO drillDone,1;
WaitUntil drillDone = 0;
        MoveL RelTool(Target_1510,0,0,-10),v30,z10,DrillTool\WObj:=FakeWing;
        MoveL RelTool(Target_1520,0,0,-10),v30,z10,DrillTool\WObj:=FakeWing;
        MoveL Target_1520,v30,fine,DrillTool\WObj:=FakeWing;
SetDO drillDone,1;
WaitUntil drillDone = 0;
        MoveL RelTool(Target_1520,0,0,-10),v30,z10,DrillTool\WObj:=FakeWing;
        MoveL RelTool(Target_1530,0,0,-10),v30,z10,DrillTool\WObj:=FakeWing;
        MoveL Target_1530,v30,fine,DrillTool\WObj:=FakeWing;
SetDO drillDone,1;
WaitUntil drillDone = 0;
        MoveL RelTool(Target_1530,0,0,-10),v30,z10,DrillTool\WObj:=FakeWing;
        MoveL RelTool(Target_1540,0,0,-10),v30,z10,DrillTool\WObj:=FakeWing;
        MoveL Target_1540,v30,fine,DrillTool\WObj:=FakeWing;
SetDO drillDone,1;
WaitUntil drillDone = 0;
        MoveL RelTool(Target_1540,0,0,-10),v30,z10,DrillTool\WObj:=FakeWing;
        MoveL RelTool(Target_1550,0,0,-10),v30,z10,DrillTool\WObj:=FakeWing;
        MoveL Target_1550,v30,fine,DrillTool\WObj:=FakeWing;
SetDO drillDone,1;
WaitUntil drillDone = 0;
        MoveL RelTool(Target_1550,0,0,-10),v30,z10,DrillTool\WObj:=FakeWing;
        MoveL RelTool(Target_1560,0,0,-10),v30,z10,DrillTool\WObj:=FakeWing;
        MoveL Target_1560,v30,fine,DrillTool\WObj:=FakeWing;
SetDO drillDone,1;
WaitUntil drillDone = 0;
        MoveL RelTool(Target_1560,0,0,-10),v30,z10,DrillTool\WObj:=FakeWing;
        MoveL RelTool(Target_1570,0,0,-10),v30,z10,DrillTool\WObj:=FakeWing;
        MoveL Target_1570,v30,fine,DrillTool\WObj:=FakeWing;
SetDO drillDone,1;
WaitUntil drillDone = 0;
        MoveL RelTool(Target_1570,0,0,-10),v30,z10,DrillTool\WObj:=FakeWing;
        MoveL RelTool(Target_1580,0,0,-10),v30,z10,DrillTool\WObj:=FakeWing;
        MoveL Target_1580,v30,fine,DrillTool\WObj:=FakeWing;
SetDO drillDone,1;
WaitUntil drillDone = 0;
        MoveL RelTool(Target_1580,0,0,-10),v30,z10,DrillTool\WObj:=FakeWing;
        MoveL RelTool(Target_1590,0,0,-10),v30,z10,DrillTool\WObj:=FakeWing;
        MoveL Target_1590,v30,fine,DrillTool\WObj:=FakeWing;
SetDO drillDone,1;
WaitUntil drillDone = 0;
        MoveL RelTool(Target_1590,0,0,-10),v30,z10,DrillTool\WObj:=FakeWing;
        MoveL RelTool(Target_1600,0,0,-10),v30,z10,DrillTool\WObj:=FakeWing;
        MoveL Target_1600,v30,fine,DrillTool\WObj:=FakeWing;
SetDO drillDone,1;
WaitUntil drillDone = 0;
        MoveL RelTool(Target_1600,0,0,-10),v30,z10,DrillTool\WObj:=FakeWing;
        MoveL RelTool(Target_1610,0,0,-10),v30,z10,DrillTool\WObj:=FakeWing;
        MoveL Target_1610,v30,fine,DrillTool\WObj:=FakeWing;
SetDO drillDone,1;
WaitUntil drillDone = 0;
        MoveL RelTool(Target_1610,0,0,-10),v30,z10,DrillTool\WObj:=FakeWing;
        MoveL RelTool(Target_1620,0,0,-10),v30,z10,DrillTool\WObj:=FakeWing;
        MoveL Target_1620,v30,fine,DrillTool\WObj:=FakeWing;
SetDO drillDone,1;
WaitUntil drillDone = 0;
        MoveL RelTool(Target_1620,0,0,-10),v30,z10,DrillTool\WObj:=FakeWing;
        MoveL RelTool(Target_1630,0,0,-10),v30,z10,DrillTool\WObj:=FakeWing;
        MoveL Target_1630,v30,fine,DrillTool\WObj:=FakeWing;
SetDO drillDone,1;
WaitUntil drillDone = 0;
        MoveL RelTool(Target_1630,0,0,-10),v30,z10,DrillTool\WObj:=FakeWing;
        MoveL RelTool(Target_1640,0,0,-10),v30,z10,DrillTool\WObj:=FakeWing;
        MoveL Target_1640,v30,fine,DrillTool\WObj:=FakeWing;
SetDO drillDone,1;
WaitUntil drillDone = 0;
        MoveL RelTool(Target_1640,0,0,-10),v30,z10,DrillTool\WObj:=FakeWing;
        MoveL RelTool(Target_1650,0,0,-10),v30,z10,DrillTool\WObj:=FakeWing;
        MoveL Target_1650,v30,fine,DrillTool\WObj:=FakeWing;
SetDO drillDone,1;
WaitUntil drillDone = 0;
        MoveL RelTool(Target_1650,0,0,-10),v30,z10,DrillTool\WObj:=FakeWing;
        MoveL RelTool(Target_1660,0,0,-10),v30,z10,DrillTool\WObj:=FakeWing;
        MoveL Target_1660,v30,fine,DrillTool\WObj:=FakeWing;
SetDO drillDone,1;
WaitUntil drillDone = 0;
        MoveL RelTool(Target_1660,0,0,-10),v30,z10,DrillTool\WObj:=FakeWing;
        MoveL RelTool(Target_1670,0,0,-10),v30,z10,DrillTool\WObj:=FakeWing;
        MoveL Target_1670,v30,fine,DrillTool\WObj:=FakeWing;
SetDO drillDone,1;
WaitUntil drillDone = 0;
        MoveL RelTool(Target_1670,0,0,-10),v30,z10,DrillTool\WObj:=FakeWing;
        MoveL RelTool(Target_1680,0,0,-10),v30,z10,DrillTool\WObj:=FakeWing;
        MoveL Target_1680,v30,fine,DrillTool\WObj:=FakeWing;
SetDO drillDone,1;
WaitUntil drillDone = 0;
        MoveL RelTool(Target_1680,0,0,-10),v30,z10,DrillTool\WObj:=FakeWing;
        MoveL RelTool(Target_1690,0,0,-10),v30,z10,DrillTool\WObj:=FakeWing;
        MoveL Target_1690,v30,fine,DrillTool\WObj:=FakeWing;
SetDO drillDone,1;
WaitUntil drillDone = 0;
        MoveL RelTool(Target_1690,0,0,-10),v30,z10,DrillTool\WObj:=FakeWing;
        MoveL RelTool(Target_1700,0,0,-10),v30,z10,DrillTool\WObj:=FakeWing;
        MoveL Target_1700,v30,fine,DrillTool\WObj:=FakeWing;
SetDO drillDone,1;
WaitUntil drillDone = 0;
        MoveL RelTool(Target_1700,0,0,-10),v30,z10,DrillTool\WObj:=FakeWing;
        MoveL RelTool(Target_1710,0,0,-10),v30,z10,DrillTool\WObj:=FakeWing;
        MoveL Target_1710,v30,fine,DrillTool\WObj:=FakeWing;
SetDO drillDone,1;
WaitUntil drillDone = 0;
        MoveL RelTool(Target_1710,0,0,-10),v30,z10,DrillTool\WObj:=FakeWing;
        MoveL RelTool(Target_1720,0,0,-10),v30,z10,DrillTool\WObj:=FakeWing;
        MoveL Target_1720,v30,fine,DrillTool\WObj:=FakeWing;
SetDO drillDone,1;
WaitUntil drillDone = 0;
        MoveL RelTool(Target_1720,0,0,-10),v30,z10,DrillTool\WObj:=FakeWing;
        MoveL RelTool(Target_1730,0,0,-10),v30,z10,DrillTool\WObj:=FakeWing;
        MoveL Target_1730,v30,fine,DrillTool\WObj:=FakeWing;
SetDO drillDone,1;
WaitUntil drillDone = 0;
        MoveL RelTool(Target_1730,0,0,-10),v30,z10,DrillTool\WObj:=FakeWing;
        MoveL RelTool(Target_1740,0,0,-10),v30,z10,DrillTool\WObj:=FakeWing;
        MoveL Target_1740,v30,fine,DrillTool\WObj:=FakeWing;
SetDO drillDone,1;
WaitUntil drillDone = 0;
        MoveL RelTool(Target_1740,0,0,-10),v30,z10,DrillTool\WObj:=FakeWing;
        MoveL RelTool(Target_1750,0,0,-10),v30,z10,DrillTool\WObj:=FakeWing;
        MoveL Target_1750,v30,fine,DrillTool\WObj:=FakeWing;
SetDO drillDone,1;
WaitUntil drillDone = 0;
        MoveL RelTool(Target_1750,0,0,-10),v30,z10,DrillTool\WObj:=FakeWing;
        MoveL RelTool(Target_1760,0,0,-10),v30,z10,DrillTool\WObj:=FakeWing;
        MoveL Target_1760,v30,fine,DrillTool\WObj:=FakeWing;
SetDO drillDone,1;
WaitUntil drillDone = 0;
        MoveL RelTool(Target_1760,0,0,-10),v30,z10,DrillTool\WObj:=FakeWing;
        MoveL RelTool(Target_1770,0,0,-10),v30,z10,DrillTool\WObj:=FakeWing;
        MoveL Target_1770,v30,fine,DrillTool\WObj:=FakeWing;
SetDO drillDone,1;
WaitUntil drillDone = 0;
        MoveL RelTool(Target_1770,0,0,-10),v30,z10,DrillTool\WObj:=FakeWing;
        MoveL RelTool(Target_1780,0,0,-10),v30,z10,DrillTool\WObj:=FakeWing;
        MoveL Target_1780,v30,fine,DrillTool\WObj:=FakeWing;
SetDO drillDone,1;
WaitUntil drillDone = 0;
        MoveL RelTool(Target_1780,0,0,-10),v30,z10,DrillTool\WObj:=FakeWing;
        MoveL RelTool(Target_1790,0,0,-10),v30,z10,DrillTool\WObj:=FakeWing;
        MoveL Target_1790,v30,fine,DrillTool\WObj:=FakeWing;
SetDO drillDone,1;
WaitUntil drillDone = 0;
        MoveL RelTool(Target_1790,0,0,-10),v30,z10,DrillTool\WObj:=FakeWing;
        MoveL RelTool(Target_1800,0,0,-10),v30,z10,DrillTool\WObj:=FakeWing;
        MoveL Target_1800,v30,fine,DrillTool\WObj:=FakeWing;
SetDO drillDone,1;
WaitUntil drillDone = 0;
        MoveL RelTool(Target_1800,0,0,-10),v30,z10,DrillTool\WObj:=FakeWing;
        MoveL RelTool(Target_1810,0,0,-10),v30,z10,DrillTool\WObj:=FakeWing;
        MoveL Target_1810,v30,fine,DrillTool\WObj:=FakeWing;
SetDO drillDone,1;
WaitUntil drillDone = 0;
        MoveL RelTool(Target_1810,0,0,-10),v30,z10,DrillTool\WObj:=FakeWing;
        MoveL RelTool(Target_1820,0,0,-10),v30,z10,DrillTool\WObj:=FakeWing;
        MoveL Target_1820,v30,fine,DrillTool\WObj:=FakeWing;
SetDO drillDone,1;
WaitUntil drillDone = 0;
        MoveL RelTool(Target_1820,0,0,-10),v30,z10,DrillTool\WObj:=FakeWing;
        MoveL RelTool(Target_1830,0,0,-10),v30,z10,DrillTool\WObj:=FakeWing;
        MoveL Target_1830,v30,fine,DrillTool\WObj:=FakeWing;
SetDO drillDone,1;
WaitUntil drillDone = 0;
        MoveL RelTool(Target_1830,0,0,-10),v30,z10,DrillTool\WObj:=FakeWing;
        MoveL RelTool(Target_1840,0,0,-10),v30,z10,DrillTool\WObj:=FakeWing;
        MoveL Target_1840,v30,fine,DrillTool\WObj:=FakeWing;
SetDO drillDone,1;
WaitUntil drillDone = 0;
        MoveL RelTool(Target_1840,0,0,-10),v30,z10,DrillTool\WObj:=FakeWing;
        MoveL RelTool(Target_1850,0,0,-10),v30,z10,DrillTool\WObj:=FakeWing;
        MoveL Target_1850,v30,fine,DrillTool\WObj:=FakeWing;
SetDO drillDone,1;
WaitUntil drillDone = 0;
        MoveL RelTool(Target_1850,0,0,-10),v30,z10,DrillTool\WObj:=FakeWing;
        MoveL RelTool(Target_1860,0,0,-10),v30,z10,DrillTool\WObj:=FakeWing;
        MoveL Target_1860,v30,fine,DrillTool\WObj:=FakeWing;
SetDO drillDone,1;
WaitUntil drillDone = 0;
        MoveL RelTool(Target_1860,0,0,-10),v30,z10,DrillTool\WObj:=FakeWing;
        MoveL RelTool(Target_1870,0,0,-10),v30,z10,DrillTool\WObj:=FakeWing;
        MoveL Target_1870,v30,fine,DrillTool\WObj:=FakeWing;
SetDO drillDone,1;
WaitUntil drillDone = 0;
        MoveL RelTool(Target_1870,0,0,-10),v30,z10,DrillTool\WObj:=FakeWing;
        MoveL RelTool(Target_1880,0,0,-10),v30,z10,DrillTool\WObj:=FakeWing;
        MoveL Target_1880,v30,fine,DrillTool\WObj:=FakeWing;
SetDO drillDone,1;
WaitUntil drillDone = 0;
        MoveL RelTool(Target_1880,0,0,-10),v30,z10,DrillTool\WObj:=FakeWing;
        MoveL RelTool(Target_1890,0,0,-10),v30,z10,DrillTool\WObj:=FakeWing;
        MoveL Target_1890,v30,fine,DrillTool\WObj:=FakeWing;
SetDO drillDone,1;
WaitUntil drillDone = 0;
        MoveL RelTool(Target_1890,0,0,-10),v30,z10,DrillTool\WObj:=FakeWing;
        MoveL RelTool(Target_1900,0,0,-10),v30,z10,DrillTool\WObj:=FakeWing;
        MoveL Target_1900,v30,fine,DrillTool\WObj:=FakeWing;
SetDO drillDone,1;
WaitUntil drillDone = 0;
        MoveL RelTool(Target_1900,0,0,-10),v30,z10,DrillTool\WObj:=FakeWing;
        MoveL RelTool(Target_1910,0,0,-10),v30,z10,DrillTool\WObj:=FakeWing;
        MoveL Target_1910,v30,fine,DrillTool\WObj:=FakeWing;
SetDO drillDone,1;
WaitUntil drillDone = 0;
        MoveL RelTool(Target_1910,0,0,-10),v30,z10,DrillTool\WObj:=FakeWing;
        MoveL RelTool(Target_1920,0,0,-10),v30,z10,DrillTool\WObj:=FakeWing;
        MoveL Target_1920,v30,fine,DrillTool\WObj:=FakeWing;
SetDO drillDone,1;
WaitUntil drillDone = 0;
        MoveL RelTool(Target_1920,0,0,-10),v30,z10,DrillTool\WObj:=FakeWing;
        MoveL RelTool(Target_1930,0,0,-10),v30,z10,DrillTool\WObj:=FakeWing;
        MoveL Target_1930,v30,fine,DrillTool\WObj:=FakeWing;
SetDO drillDone,1;
WaitUntil drillDone = 0;
        MoveL RelTool(Target_1930,0,0,-10),v30,z10,DrillTool\WObj:=FakeWing;
        MoveL RelTool(Target_1940,0,0,-10),v30,z10,DrillTool\WObj:=FakeWing;
        MoveL Target_1940,v30,fine,DrillTool\WObj:=FakeWing;
SetDO drillDone,1;
WaitUntil drillDone = 0;
        MoveL RelTool(Target_1940,0,0,-10),v30,z10,DrillTool\WObj:=FakeWing;
        MoveL RelTool(Target_1950,0,0,-10),v30,z10,DrillTool\WObj:=FakeWing;
        MoveL Target_1950,v30,fine,DrillTool\WObj:=FakeWing;
SetDO drillDone,1;
WaitUntil drillDone = 0;
        MoveL RelTool(Target_1950,0,0,-10),v30,z10,DrillTool\WObj:=FakeWing;
        MoveL RelTool(Target_1960,0,0,-10),v30,z10,DrillTool\WObj:=FakeWing;
        MoveL Target_1960,v30,fine,DrillTool\WObj:=FakeWing;
SetDO drillDone,1;
WaitUntil drillDone = 0;
        MoveL RelTool(Target_1960,0,0,-10),v30,z10,DrillTool\WObj:=FakeWing;
        MoveL RelTool(Target_1970,0,0,-10),v30,z10,DrillTool\WObj:=FakeWing;
        MoveL Target_1970,v30,fine,DrillTool\WObj:=FakeWing;
SetDO drillDone,1;
WaitUntil drillDone = 0;
        MoveL RelTool(Target_1970,0,0,-10),v30,z10,DrillTool\WObj:=FakeWing;
        MoveL RelTool(Target_1980,0,0,-10),v30,z10,DrillTool\WObj:=FakeWing;
        MoveL Target_1980,v30,fine,DrillTool\WObj:=FakeWing;
SetDO drillDone,1;
WaitUntil drillDone = 0;
        MoveL RelTool(Target_1980,0,0,-10),v30,z10,DrillTool\WObj:=FakeWing;
        MoveL RelTool(Target_1990,0,0,-10),v30,z10,DrillTool\WObj:=FakeWing;
        MoveL Target_1990,v30,fine,DrillTool\WObj:=FakeWing;
SetDO drillDone,1;
WaitUntil drillDone = 0;
        MoveL RelTool(Target_1990,0,0,-10),v30,z10,DrillTool\WObj:=FakeWing;
        MoveL RelTool(Target_2000,0,0,-10),v30,z10,DrillTool\WObj:=FakeWing;
        MoveL Target_2000,v30,fine,DrillTool\WObj:=FakeWing;
SetDO drillDone,1;
WaitUntil drillDone = 0;
        MoveL RelTool(Target_2000,0,0,-10),v30,z10,DrillTool\WObj:=FakeWing;
        MoveL RelTool(Target_2010,0,0,-10),v30,z10,DrillTool\WObj:=FakeWing;
        MoveL Target_2010,v30,fine,DrillTool\WObj:=FakeWing;
SetDO drillDone,1;
WaitUntil drillDone = 0;
        MoveL RelTool(Target_2010,0,0,-10),v30,z10,DrillTool\WObj:=FakeWing;
        MoveL RelTool(Target_2020,0,0,-10),v30,z10,DrillTool\WObj:=FakeWing;
        MoveL Target_2020,v30,fine,DrillTool\WObj:=FakeWing;
SetDO drillDone,1;
WaitUntil drillDone = 0;
        MoveL RelTool(Target_2020,0,0,-10),v30,z10,DrillTool\WObj:=FakeWing;
        MoveL RelTool(Target_2030,0,0,-10),v30,z10,DrillTool\WObj:=FakeWing;
        MoveL Target_2030,v30,fine,DrillTool\WObj:=FakeWing;
SetDO drillDone,1;
WaitUntil drillDone = 0;
        MoveL RelTool(Target_2030,0,0,-10),v30,z10,DrillTool\WObj:=FakeWing;
        MoveL RelTool(Target_2040,0,0,-10),v30,z10,DrillTool\WObj:=FakeWing;
        MoveL Target_2040,v30,fine,DrillTool\WObj:=FakeWing;
SetDO drillDone,1;
WaitUntil drillDone = 0;
        MoveL RelTool(Target_2040,0,0,-10),v30,z10,DrillTool\WObj:=FakeWing;
        MoveL RelTool(Target_2050,0,0,-10),v30,z10,DrillTool\WObj:=FakeWing;
        MoveL Target_2050,v30,fine,DrillTool\WObj:=FakeWing;
SetDO drillDone,1;
WaitUntil drillDone = 0;
        MoveL RelTool(Target_2050,0,0,-10),v30,z10,DrillTool\WObj:=FakeWing;
        MoveL RelTool(Target_2060,0,0,-10),v30,z10,DrillTool\WObj:=FakeWing;
        MoveL Target_2060,v30,fine,DrillTool\WObj:=FakeWing;
SetDO drillDone,1;
WaitUntil drillDone = 0;
        MoveL RelTool(Target_2060,0,0,-10),v30,z10,DrillTool\WObj:=FakeWing;
        MoveL RelTool(Target_2070,0,0,-10),v30,z10,DrillTool\WObj:=FakeWing;
        MoveL Target_2070,v30,fine,DrillTool\WObj:=FakeWing;
SetDO drillDone,1;
WaitUntil drillDone = 0;
        MoveL RelTool(Target_2070,0,0,-10),v30,z10,DrillTool\WObj:=FakeWing;
        MoveL RelTool(Target_2080,0,0,-10),v30,z10,DrillTool\WObj:=FakeWing;
        MoveL Target_2080,v30,fine,DrillTool\WObj:=FakeWing;
SetDO drillDone,1;
WaitUntil drillDone = 0;
        MoveL RelTool(Target_2080,0,0,-10),v30,z10,DrillTool\WObj:=FakeWing;
        MoveL RelTool(Target_2090,0,0,-10),v30,z10,DrillTool\WObj:=FakeWing;
        MoveL Target_2090,v30,fine,DrillTool\WObj:=FakeWing;
SetDO drillDone,1;
WaitUntil drillDone = 0;
        MoveL RelTool(Target_2090,0,0,-10),v30,z10,DrillTool\WObj:=FakeWing;
        MoveL RelTool(Target_2100,0,0,-10),v30,z10,DrillTool\WObj:=FakeWing;
        MoveL Target_2100,v30,fine,DrillTool\WObj:=FakeWing;
SetDO drillDone,1;
WaitUntil drillDone = 0;
        MoveL RelTool(Target_2100,0,0,-10),v30,z10,DrillTool\WObj:=FakeWing;
        MoveL RelTool(Target_2110,0,0,-10),v30,z10,DrillTool\WObj:=FakeWing;
        MoveL Target_2110,v30,fine,DrillTool\WObj:=FakeWing;
SetDO drillDone,1;
WaitUntil drillDone = 0;
        MoveL RelTool(Target_2110,0,0,-10),v30,z10,DrillTool\WObj:=FakeWing;
        MoveL RelTool(Target_2120,0,0,-10),v30,z10,DrillTool\WObj:=FakeWing;
        MoveL Target_2120,v30,fine,DrillTool\WObj:=FakeWing;
SetDO drillDone,1;
WaitUntil drillDone = 0;
        MoveL RelTool(Target_2120,0,0,-10),v30,z10,DrillTool\WObj:=FakeWing;
        MoveL RelTool(Target_2130,0,0,-10),v30,z10,DrillTool\WObj:=FakeWing;
        MoveL Target_2130,v30,fine,DrillTool\WObj:=FakeWing;
SetDO drillDone,1;
WaitUntil drillDone = 0;
        MoveL RelTool(Target_2130,0,0,-10),v30,z10,DrillTool\WObj:=FakeWing;
        MoveL RelTool(Target_2140,0,0,-10),v30,z10,DrillTool\WObj:=FakeWing;
        MoveL Target_2140,v30,fine,DrillTool\WObj:=FakeWing;
SetDO drillDone,1;
WaitUntil drillDone = 0;
        MoveL RelTool(Target_2140,0,0,-10),v30,z10,DrillTool\WObj:=FakeWing;
        MoveL RelTool(Target_2150,0,0,-10),v30,z10,DrillTool\WObj:=FakeWing;
        MoveL Target_2150,v30,fine,DrillTool\WObj:=FakeWing;
SetDO drillDone,1;
WaitUntil drillDone = 0;
        MoveL RelTool(Target_2150,0,0,-10),v30,z10,DrillTool\WObj:=FakeWing;
        MoveL RelTool(Target_2160,0,0,-10),v30,z10,DrillTool\WObj:=FakeWing;
        MoveL Target_2160,v30,fine,DrillTool\WObj:=FakeWing;
SetDO drillDone,1;
WaitUntil drillDone = 0;
        MoveL RelTool(Target_2160,0,0,-10),v30,z10,DrillTool\WObj:=FakeWing;
        MoveL RelTool(Target_2170,0,0,-10),v30,z10,DrillTool\WObj:=FakeWing;
        MoveL Target_2170,v30,fine,DrillTool\WObj:=FakeWing;
SetDO drillDone,1;
WaitUntil drillDone = 0;
        MoveL RelTool(Target_2170,0,0,-10),v30,z10,DrillTool\WObj:=FakeWing;
        MoveL RelTool(Target_2180,0,0,-10),v30,z10,DrillTool\WObj:=FakeWing;
        MoveL Target_2180,v30,fine,DrillTool\WObj:=FakeWing;
SetDO drillDone,1;
WaitUntil drillDone = 0;
        MoveL RelTool(Target_2180,0,0,-10),v30,z10,DrillTool\WObj:=FakeWing;
        MoveL RelTool(Target_2190,0,0,-10),v30,z10,DrillTool\WObj:=FakeWing;
        MoveL Target_2190,v30,fine,DrillTool\WObj:=FakeWing;
SetDO drillDone,1;
WaitUntil drillDone = 0;
        MoveL RelTool(Target_2190,0,0,-10),v30,z10,DrillTool\WObj:=FakeWing;
        MoveL RelTool(Target_2200,0,0,-10),v30,z10,DrillTool\WObj:=FakeWing;
        MoveL Target_2200,v30,fine,DrillTool\WObj:=FakeWing;
SetDO drillDone,1;
WaitUntil drillDone = 0;
        MoveL RelTool(Target_2200,0,0,-10),v30,z10,DrillTool\WObj:=FakeWing;
        MoveL RelTool(Target_2210,0,0,-10),v30,z10,DrillTool\WObj:=FakeWing;
        MoveL Target_2210,v30,fine,DrillTool\WObj:=FakeWing;
SetDO drillDone,1;
WaitUntil drillDone = 0;
        MoveL RelTool(Target_2210,0,0,-10),v30,z10,DrillTool\WObj:=FakeWing;
        MoveL RelTool(Target_2220,0,0,-10),v30,z10,DrillTool\WObj:=FakeWing;
        MoveL Target_2220,v30,fine,DrillTool\WObj:=FakeWing;
SetDO drillDone,1;
WaitUntil drillDone = 0;
        MoveL RelTool(Target_2220,0,0,-10),v30,z10,DrillTool\WObj:=FakeWing;
        MoveL RelTool(Target_2230,0,0,-10),v30,z10,DrillTool\WObj:=FakeWing;
        MoveL Target_2230,v30,fine,DrillTool\WObj:=FakeWing;
SetDO drillDone,1;
WaitUntil drillDone = 0;
        MoveL RelTool(Target_2230,0,0,-10),v30,z10,DrillTool\WObj:=FakeWing;
        MoveL RelTool(Target_2240,0,0,-10),v30,z10,DrillTool\WObj:=FakeWing;
        MoveL Target_2240,v30,fine,DrillTool\WObj:=FakeWing;
SetDO drillDone,1;
WaitUntil drillDone = 0;
        MoveL RelTool(Target_2240,0,0,-10),v30,z10,DrillTool\WObj:=FakeWing;
        MoveL RelTool(Target_2250,0,0,-10),v30,z10,DrillTool\WObj:=FakeWing;
        MoveL Target_2250,v30,fine,DrillTool\WObj:=FakeWing;
SetDO drillDone,1;
WaitUntil drillDone = 0;
        MoveL RelTool(Target_2250,0,0,-10),v30,z10,DrillTool\WObj:=FakeWing;
        MoveL RelTool(Target_2260,0,0,-10),v30,z10,DrillTool\WObj:=FakeWing;
        MoveL Target_2260,v30,fine,DrillTool\WObj:=FakeWing;
SetDO drillDone,1;
WaitUntil drillDone = 0;
        MoveL RelTool(Target_2260,0,0,-10),v30,z10,DrillTool\WObj:=FakeWing;
        MoveL RelTool(Target_2270,0,0,-10),v30,z10,DrillTool\WObj:=FakeWing;
        MoveL Target_2270,v30,fine,DrillTool\WObj:=FakeWing;
SetDO drillDone,1;
WaitUntil drillDone = 0;
        MoveL RelTool(Target_2270,0,0,-10),v30,z10,DrillTool\WObj:=FakeWing;
        MoveL RelTool(Target_2280,0,0,-10),v30,z10,DrillTool\WObj:=FakeWing;
        MoveL Target_2280,v30,fine,DrillTool\WObj:=FakeWing;
SetDO drillDone,1;
WaitUntil drillDone = 0;
        MoveL RelTool(Target_2280,0,0,-10),v30,z10,DrillTool\WObj:=FakeWing;
        MoveL RelTool(Target_2290,0,0,-10),v30,z10,DrillTool\WObj:=FakeWing;
        MoveL Target_2290,v30,fine,DrillTool\WObj:=FakeWing;
SetDO drillDone,1;
WaitUntil drillDone = 0;
        MoveL RelTool(Target_2290,0,0,-10),v30,z10,DrillTool\WObj:=FakeWing;
        MoveL RelTool(Target_2300,0,0,-10),v30,z10,DrillTool\WObj:=FakeWing;
        MoveL Target_2300,v30,fine,DrillTool\WObj:=FakeWing;
SetDO drillDone,1;
WaitUntil drillDone = 0;
        MoveL RelTool(Target_2300,0,0,-10),v30,z10,DrillTool\WObj:=FakeWing;
        MoveL RelTool(Target_2310,0,0,-10),v30,z10,DrillTool\WObj:=FakeWing;
        MoveL Target_2310,v30,fine,DrillTool\WObj:=FakeWing;
SetDO drillDone,1;
WaitUntil drillDone = 0;
        MoveL RelTool(Target_2310,0,0,-10),v30,z10,DrillTool\WObj:=FakeWing;
        MoveL RelTool(Target_2320,0,0,-10),v30,z10,DrillTool\WObj:=FakeWing;
        MoveL Target_2320,v30,fine,DrillTool\WObj:=FakeWing;
SetDO drillDone,1;
WaitUntil drillDone = 0;
        MoveL RelTool(Target_2320,0,0,-10),v30,z10,DrillTool\WObj:=FakeWing;
        MoveL RelTool(Target_2330,0,0,-10),v30,z10,DrillTool\WObj:=FakeWing;
        MoveL Target_2330,v30,fine,DrillTool\WObj:=FakeWing;
SetDO drillDone,1;
WaitUntil drillDone = 0;
        MoveL RelTool(Target_2330,0,0,-10),v30,z10,DrillTool\WObj:=FakeWing;
        MoveL RelTool(Target_2340,0,0,-10),v30,z10,DrillTool\WObj:=FakeWing;
        MoveL Target_2340,v30,fine,DrillTool\WObj:=FakeWing;
SetDO drillDone,1;
WaitUntil drillDone = 0;
        MoveL RelTool(Target_2340,0,0,-10),v30,z10,DrillTool\WObj:=FakeWing;
        MoveL RelTool(Target_2350,0,0,-10),v30,z10,DrillTool\WObj:=FakeWing;
        MoveL Target_2350,v30,fine,DrillTool\WObj:=FakeWing;
SetDO drillDone,1;
WaitUntil drillDone = 0;
        MoveL RelTool(Target_2350,0,0,-10),v30,z10,DrillTool\WObj:=FakeWing;
        MoveL RelTool(Target_2360,0,0,-10),v30,z10,DrillTool\WObj:=FakeWing;
        MoveL Target_2360,v30,fine,DrillTool\WObj:=FakeWing;
SetDO drillDone,1;
WaitUntil drillDone = 0;
        MoveL RelTool(Target_2360,0,0,-10),v30,z10,DrillTool\WObj:=FakeWing;
        MoveL RelTool(Target_2370,0,0,-10),v30,z10,DrillTool\WObj:=FakeWing;
        MoveL Target_2370,v30,fine,DrillTool\WObj:=FakeWing;
SetDO drillDone,1;
WaitUntil drillDone = 0;
        MoveL RelTool(Target_2370,0,0,-10),v30,z10,DrillTool\WObj:=FakeWing;
        MoveL RelTool(Target_2380,0,0,-10),v30,z10,DrillTool\WObj:=FakeWing;
        MoveL Target_2380,v30,fine,DrillTool\WObj:=FakeWing;
SetDO drillDone,1;
WaitUntil drillDone = 0;
        MoveL RelTool(Target_2380,0,0,-10),v30,z10,DrillTool\WObj:=FakeWing;
        MoveL RelTool(Target_2390,0,0,-10),v30,z10,DrillTool\WObj:=FakeWing;
        MoveL Target_2390,v30,fine,DrillTool\WObj:=FakeWing;
SetDO drillDone,1;
WaitUntil drillDone = 0;
        MoveL RelTool(Target_2390,0,0,-10),v30,z10,DrillTool\WObj:=FakeWing;
        MoveL RelTool(Target_2400,0,0,-10),v30,z10,DrillTool\WObj:=FakeWing;
        MoveL Target_2400,v30,fine,DrillTool\WObj:=FakeWing;
SetDO drillDone,1;
WaitUntil drillDone = 0;
        MoveL RelTool(Target_2400,0,0,-10),v30,z10,DrillTool\WObj:=FakeWing;
        MoveL RelTool(Target_2410,0,0,-10),v30,z10,DrillTool\WObj:=FakeWing;
        MoveL Target_2410,v30,fine,DrillTool\WObj:=FakeWing;
SetDO drillDone,1;
WaitUntil drillDone = 0;
        MoveL RelTool(Target_2410,0,0,-10),v30,z10,DrillTool\WObj:=FakeWing;
        MoveL RelTool(Target_2420,0,0,-10),v30,z10,DrillTool\WObj:=FakeWing;
        MoveL Target_2420,v30,fine,DrillTool\WObj:=FakeWing;
SetDO drillDone,1;
WaitUntil drillDone = 0;
        MoveL RelTool(Target_2420,0,0,-10),v30,z10,DrillTool\WObj:=FakeWing;
        MoveL RelTool(Target_2430,0,0,-10),v30,z10,DrillTool\WObj:=FakeWing;
        MoveL Target_2430,v30,fine,DrillTool\WObj:=FakeWing;
SetDO drillDone,1;
WaitUntil drillDone = 0;
        MoveL RelTool(Target_2430,0,0,-10),v30,z10,DrillTool\WObj:=FakeWing;
        MoveL RelTool(Target_2440,0,0,-10),v30,z10,DrillTool\WObj:=FakeWing;
        MoveL Target_2440,v30,fine,DrillTool\WObj:=FakeWing;
SetDO drillDone,1;
WaitUntil drillDone = 0;
        MoveL RelTool(Target_2440,0,0,-10),v30,z10,DrillTool\WObj:=FakeWing;
        MoveL RelTool(Target_2450,0,0,-10),v30,z10,DrillTool\WObj:=FakeWing;
        MoveL Target_2450,v30,fine,DrillTool\WObj:=FakeWing;
SetDO drillDone,1;
WaitUntil drillDone = 0;
        MoveL RelTool(Target_2450,0,0,-10),v30,z10,DrillTool\WObj:=FakeWing;
        MoveL RelTool(Target_2460,0,0,-10),v30,z10,DrillTool\WObj:=FakeWing;
        MoveL Target_2460,v30,fine,DrillTool\WObj:=FakeWing;
SetDO drillDone,1;
WaitUntil drillDone = 0;
        MoveL RelTool(Target_2460,0,0,-10),v30,z10,DrillTool\WObj:=FakeWing;
        MoveL RelTool(Target_2470,0,0,-10),v30,z10,DrillTool\WObj:=FakeWing;
        MoveL Target_2470,v30,fine,DrillTool\WObj:=FakeWing;
SetDO drillDone,1;
WaitUntil drillDone = 0;
        MoveL RelTool(Target_2470,0,0,-10),v30,z10,DrillTool\WObj:=FakeWing;
        MoveL RelTool(Target_2480,0,0,-10),v30,z10,DrillTool\WObj:=FakeWing;
        MoveL Target_2480,v30,fine,DrillTool\WObj:=FakeWing;
SetDO drillDone,1;
WaitUntil drillDone = 0;
        MoveL RelTool(Target_2480,0,0,-10),v30,z10,DrillTool\WObj:=FakeWing;
        MoveL RelTool(Target_2490,0,0,-10),v30,z10,DrillTool\WObj:=FakeWing;
        MoveL Target_2490,v30,fine,DrillTool\WObj:=FakeWing;
SetDO drillDone,1;
WaitUntil drillDone = 0;
        MoveL RelTool(Target_2490,0,0,-10),v30,z10,DrillTool\WObj:=FakeWing;
        MoveL RelTool(Target_2500,0,0,-10),v30,z10,DrillTool\WObj:=FakeWing;
        MoveL Target_2500,v30,fine,DrillTool\WObj:=FakeWing;
SetDO drillDone,1;
WaitUntil drillDone = 0;
        MoveL RelTool(Target_2500,0,0,-10),v30,z10,DrillTool\WObj:=FakeWing;
        MoveL RelTool(Target_2510,0,0,-10),v30,z10,DrillTool\WObj:=FakeWing;
        MoveL Target_2510,v30,fine,DrillTool\WObj:=FakeWing;
SetDO drillDone,1;
WaitUntil drillDone = 0;
        MoveL RelTool(Target_2510,0,0,-10),v30,z10,DrillTool\WObj:=FakeWing;
        MoveL RelTool(Target_2520,0,0,-10),v30,z10,DrillTool\WObj:=FakeWing;
        MoveL Target_2520,v30,fine,DrillTool\WObj:=FakeWing;
SetDO drillDone,1;
WaitUntil drillDone = 0;
        MoveL RelTool(Target_2520,0,0,-10),v30,z10,DrillTool\WObj:=FakeWing;
        MoveL RelTool(Target_2530,0,0,-10),v30,z10,DrillTool\WObj:=FakeWing;
        MoveL Target_2530,v30,fine,DrillTool\WObj:=FakeWing;
SetDO drillDone,1;
WaitUntil drillDone = 0;
        MoveL RelTool(Target_2530,0,0,-10),v30,z10,DrillTool\WObj:=FakeWing;
        MoveL RelTool(Target_2540,0,0,-10),v30,z10,DrillTool\WObj:=FakeWing;
        MoveL Target_2540,v30,fine,DrillTool\WObj:=FakeWing;
SetDO drillDone,1;
WaitUntil drillDone = 0;
        MoveL RelTool(Target_2540,0,0,-10),v30,z10,DrillTool\WObj:=FakeWing;
        MoveL RelTool(Target_2550,0,0,-10),v30,z10,DrillTool\WObj:=FakeWing;
        MoveL Target_2550,v30,fine,DrillTool\WObj:=FakeWing;
SetDO drillDone,1;
WaitUntil drillDone = 0;
        MoveL RelTool(Target_2550,0,0,-10),v30,z10,DrillTool\WObj:=FakeWing;
        MoveL RelTool(Target_2560,0,0,-10),v30,z10,DrillTool\WObj:=FakeWing;
        MoveL Target_2560,v30,fine,DrillTool\WObj:=FakeWing;
SetDO drillDone,1;
WaitUntil drillDone = 0;
        MoveL RelTool(Target_2560,0,0,-10),v30,z10,DrillTool\WObj:=FakeWing;
        MoveL RelTool(Target_2570,0,0,-10),v30,z10,DrillTool\WObj:=FakeWing;
        MoveL Target_2570,v30,fine,DrillTool\WObj:=FakeWing;
SetDO drillDone,1;
WaitUntil drillDone = 0;
        MoveL RelTool(Target_2570,0,0,-10),v30,z10,DrillTool\WObj:=FakeWing;
        MoveL RelTool(Target_2580,0,0,-10),v30,z10,DrillTool\WObj:=FakeWing;
        MoveL Target_2580,v30,fine,DrillTool\WObj:=FakeWing;
SetDO drillDone,1;
WaitUntil drillDone = 0;
        MoveL RelTool(Target_2580,0,0,-10),v30,z10,DrillTool\WObj:=FakeWing;
        MoveL RelTool(Target_2590,0,0,-10),v30,z10,DrillTool\WObj:=FakeWing;
        MoveL Target_2590,v30,fine,DrillTool\WObj:=FakeWing;
SetDO drillDone,1;
WaitUntil drillDone = 0;
        MoveL RelTool(Target_2590,0,0,-10),v30,z10,DrillTool\WObj:=FakeWing;
        MoveL RelTool(Target_2600,0,0,-10),v30,z10,DrillTool\WObj:=FakeWing;
        MoveL Target_2600,v30,fine,DrillTool\WObj:=FakeWing;
SetDO drillDone,1;
WaitUntil drillDone = 0;
        MoveL RelTool(Target_2600,0,0,-10),v30,z10,DrillTool\WObj:=FakeWing;
        MoveL RelTool(Target_2610,0,0,-10),v30,z10,DrillTool\WObj:=FakeWing;
        MoveL Target_2610,v30,fine,DrillTool\WObj:=FakeWing;
SetDO drillDone,1;
WaitUntil drillDone = 0;
        MoveL RelTool(Target_2610,0,0,-10),v30,z10,DrillTool\WObj:=FakeWing;
        MoveL RelTool(Target_2620,0,0,-10),v30,z10,DrillTool\WObj:=FakeWing;
        MoveL Target_2620,v30,fine,DrillTool\WObj:=FakeWing;
SetDO drillDone,1;
WaitUntil drillDone = 0;
        MoveL RelTool(Target_2620,0,0,-10),v30,z10,DrillTool\WObj:=FakeWing;
        MoveL RelTool(Target_2630,0,0,-10),v30,z10,DrillTool\WObj:=FakeWing;
        MoveL Target_2630,v30,fine,DrillTool\WObj:=FakeWing;
SetDO drillDone,1;
WaitUntil drillDone = 0;
        MoveL RelTool(Target_2630,0,0,-10),v30,z10,DrillTool\WObj:=FakeWing;
        MoveL RelTool(Target_2640,0,0,-10),v30,z10,DrillTool\WObj:=FakeWing;
        MoveL Target_2640,v30,fine,DrillTool\WObj:=FakeWing;
SetDO drillDone,1;
WaitUntil drillDone = 0;
        MoveL RelTool(Target_2640,0,0,-10),v30,z10,DrillTool\WObj:=FakeWing;
        MoveL RelTool(Target_2650,0,0,-10),v30,z10,DrillTool\WObj:=FakeWing;
        MoveL Target_2650,v30,fine,DrillTool\WObj:=FakeWing;
SetDO drillDone,1;
WaitUntil drillDone = 0;
        MoveL RelTool(Target_2650,0,0,-10),v30,z10,DrillTool\WObj:=FakeWing;
        MoveL RelTool(Target_2660,0,0,-10),v30,z10,DrillTool\WObj:=FakeWing;
        MoveL Target_2660,v30,fine,DrillTool\WObj:=FakeWing;
SetDO drillDone,1;
WaitUntil drillDone = 0;
        MoveL RelTool(Target_2660,0,0,-10),v30,z10,DrillTool\WObj:=FakeWing;
        MoveL RelTool(Target_2670,0,0,-10),v30,z10,DrillTool\WObj:=FakeWing;
        MoveL Target_2670,v30,fine,DrillTool\WObj:=FakeWing;
SetDO drillDone,1;
WaitUntil drillDone = 0;
        MoveL RelTool(Target_2670,0,0,-10),v30,z10,DrillTool\WObj:=FakeWing;
        MoveL RelTool(Target_2680,0,0,-10),v30,z10,DrillTool\WObj:=FakeWing;
        MoveL Target_2680,v30,fine,DrillTool\WObj:=FakeWing;
SetDO drillDone,1;
WaitUntil drillDone = 0;
        MoveL RelTool(Target_2680,0,0,-10),v30,z10,DrillTool\WObj:=FakeWing;
        MoveL RelTool(Target_2690,0,0,-10),v30,z10,DrillTool\WObj:=FakeWing;
        MoveL Target_2690,v30,fine,DrillTool\WObj:=FakeWing;
SetDO drillDone,1;
WaitUntil drillDone = 0;
        MoveL RelTool(Target_2690,0,0,-10),v30,z10,DrillTool\WObj:=FakeWing;
        MoveL RelTool(Target_2700,0,0,-10),v30,z10,DrillTool\WObj:=FakeWing;
        MoveL Target_2700,v30,fine,DrillTool\WObj:=FakeWing;
SetDO drillDone,1;
WaitUntil drillDone = 0;
        MoveL RelTool(Target_2700,0,0,-10),v30,z10,DrillTool\WObj:=FakeWing;
        MoveL RelTool(Target_2710,0,0,-10),v30,z10,DrillTool\WObj:=FakeWing;
        MoveL Target_2710,v30,fine,DrillTool\WObj:=FakeWing;
SetDO drillDone,1;
WaitUntil drillDone = 0;
        MoveL RelTool(Target_2710,0,0,-10),v30,z10,DrillTool\WObj:=FakeWing;
        MoveL RelTool(Target_2720,0,0,-10),v30,z10,DrillTool\WObj:=FakeWing;
        MoveL Target_2720,v30,fine,DrillTool\WObj:=FakeWing;
SetDO drillDone,1;
WaitUntil drillDone = 0;
        MoveL RelTool(Target_2720,0,0,-10),v30,z10,DrillTool\WObj:=FakeWing;
        MoveL RelTool(Target_2730,0,0,-10),v30,z10,DrillTool\WObj:=FakeWing;
        MoveL Target_2730,v30,fine,DrillTool\WObj:=FakeWing;
SetDO drillDone,1;
WaitUntil drillDone = 0;
        MoveL RelTool(Target_2730,0,0,-10),v30,z10,DrillTool\WObj:=FakeWing;
        MoveL RelTool(Target_2740,0,0,-10),v30,z10,DrillTool\WObj:=FakeWing;
        MoveL Target_2740,v30,fine,DrillTool\WObj:=FakeWing;
SetDO drillDone,1;
WaitUntil drillDone = 0;
        MoveL RelTool(Target_2740,0,0,-10),v30,z10,DrillTool\WObj:=FakeWing;
        MoveL RelTool(Target_2750,0,0,-10),v30,z10,DrillTool\WObj:=FakeWing;
        MoveL Target_2750,v30,fine,DrillTool\WObj:=FakeWing;
SetDO drillDone,1;
WaitUntil drillDone = 0;
        MoveL RelTool(Target_2750,0,0,-10),v30,z10,DrillTool\WObj:=FakeWing;
        MoveL RelTool(Target_2760,0,0,-10),v30,z10,DrillTool\WObj:=FakeWing;
        MoveL Target_2760,v30,fine,DrillTool\WObj:=FakeWing;
SetDO drillDone,1;
WaitUntil drillDone = 0;
        MoveL RelTool(Target_2760,0,0,-10),v30,z10,DrillTool\WObj:=FakeWing;
        MoveL RelTool(Target_2770,0,0,-10),v30,z10,DrillTool\WObj:=FakeWing;
        MoveL Target_2770,v30,fine,DrillTool\WObj:=FakeWing;
SetDO drillDone,1;
WaitUntil drillDone = 0;
        MoveL RelTool(Target_2770,0,0,-10),v30,z10,DrillTool\WObj:=FakeWing;
        MoveL RelTool(Target_2780,0,0,-10),v30,z10,DrillTool\WObj:=FakeWing;
        MoveL Target_2780,v30,fine,DrillTool\WObj:=FakeWing;
SetDO drillDone,1;
WaitUntil drillDone = 0;
        MoveL RelTool(Target_2780,0,0,-10),v30,z10,DrillTool\WObj:=FakeWing;
        MoveL RelTool(Target_2790,0,0,-10),v30,z10,DrillTool\WObj:=FakeWing;
        MoveL Target_2790,v30,fine,DrillTool\WObj:=FakeWing;
SetDO drillDone,1;
WaitUntil drillDone = 0;
        MoveL RelTool(Target_2790,0,0,-10),v30,z10,DrillTool\WObj:=FakeWing;
        MoveL RelTool(Target_2800,0,0,-10),v30,z10,DrillTool\WObj:=FakeWing;
        MoveL Target_2800,v30,fine,DrillTool\WObj:=FakeWing;
SetDO drillDone,1;
WaitUntil drillDone = 0;
        MoveL RelTool(Target_2800,0,0,-10),v30,z10,DrillTool\WObj:=FakeWing;
        MoveL RelTool(Target_2810,0,0,-10),v30,z10,DrillTool\WObj:=FakeWing;
        MoveL Target_2810,v30,fine,DrillTool\WObj:=FakeWing;
SetDO drillDone,1;
WaitUntil drillDone = 0;
        MoveL RelTool(Target_2810,0,0,-10),v30,z10,DrillTool\WObj:=FakeWing;
        MoveL RelTool(Target_2820,0,0,-10),v30,z10,DrillTool\WObj:=FakeWing;
        MoveL Target_2820,v30,fine,DrillTool\WObj:=FakeWing;
SetDO drillDone,1;
WaitUntil drillDone = 0;
        MoveL RelTool(Target_2820,0,0,-10),v30,z10,DrillTool\WObj:=FakeWing;
        MoveL RelTool(Target_2830,0,0,-10),v30,z10,DrillTool\WObj:=FakeWing;
        MoveL Target_2830,v30,fine,DrillTool\WObj:=FakeWing;
SetDO drillDone,1;
WaitUntil drillDone = 0;
        MoveL RelTool(Target_2830,0,0,-10),v30,z10,DrillTool\WObj:=FakeWing;
        MoveL RelTool(Target_2840,0,0,-10),v30,z10,DrillTool\WObj:=FakeWing;
        MoveL Target_2840,v30,fine,DrillTool\WObj:=FakeWing;
SetDO drillDone,1;
WaitUntil drillDone = 0;
        MoveL RelTool(Target_2840,0,0,-10),v30,z10,DrillTool\WObj:=FakeWing;
        MoveL RelTool(Target_2850,0,0,-10),v30,z10,DrillTool\WObj:=FakeWing;
        MoveL Target_2850,v30,fine,DrillTool\WObj:=FakeWing;
SetDO drillDone,1;
WaitUntil drillDone = 0;
        MoveL RelTool(Target_2850,0,0,-10),v30,z10,DrillTool\WObj:=FakeWing;
        MoveL RelTool(Target_2860,0,0,-10),v30,z10,DrillTool\WObj:=FakeWing;
        MoveL Target_2860,v30,fine,DrillTool\WObj:=FakeWing;
SetDO drillDone,1;
WaitUntil drillDone = 0;
        MoveL RelTool(Target_2860,0,0,-10),v30,z10,DrillTool\WObj:=FakeWing;
        MoveL RelTool(Target_2870,0,0,-10),v30,z10,DrillTool\WObj:=FakeWing;
        MoveL Target_2870,v30,fine,DrillTool\WObj:=FakeWing;
SetDO drillDone,1;
WaitUntil drillDone = 0;
        MoveL RelTool(Target_2870,0,0,-10),v30,z10,DrillTool\WObj:=FakeWing;
        MoveL RelTool(Target_2880,0,0,-10),v30,z10,DrillTool\WObj:=FakeWing;
        MoveL Target_2880,v30,fine,DrillTool\WObj:=FakeWing;
SetDO drillDone,1;
WaitUntil drillDone = 0;
        MoveL RelTool(Target_2880,0,0,-10),v30,z10,DrillTool\WObj:=FakeWing;
        MoveL RelTool(Target_2890,0,0,-10),v30,z10,DrillTool\WObj:=FakeWing;
        MoveL Target_2890,v30,fine,DrillTool\WObj:=FakeWing;
SetDO drillDone,1;
WaitUntil drillDone = 0;
        MoveL RelTool(Target_2890,0,0,-10),v30,z10,DrillTool\WObj:=FakeWing;
        MoveL RelTool(Target_2900,0,0,-10),v30,z10,DrillTool\WObj:=FakeWing;
        MoveL Target_2900,v30,fine,DrillTool\WObj:=FakeWing;
SetDO drillDone,1;
WaitUntil drillDone = 0;
        MoveL RelTool(Target_2900,0,0,-10),v30,z10,DrillTool\WObj:=FakeWing;
        MoveL RelTool(Target_2910,0,0,-10),v30,z10,DrillTool\WObj:=FakeWing;
        MoveL Target_2910,v30,fine,DrillTool\WObj:=FakeWing;
SetDO drillDone,1;
WaitUntil drillDone = 0;
        MoveL RelTool(Target_2910,0,0,-10),v30,z10,DrillTool\WObj:=FakeWing;
        MoveL RelTool(Target_2920,0,0,-10),v30,z10,DrillTool\WObj:=FakeWing;
        MoveL Target_2920,v30,fine,DrillTool\WObj:=FakeWing;
SetDO drillDone,1;
WaitUntil drillDone = 0;
        MoveL RelTool(Target_2920,0,0,-10),v30,z10,DrillTool\WObj:=FakeWing;
        MoveL RelTool(Target_2930,0,0,-10),v30,z10,DrillTool\WObj:=FakeWing;
        MoveL Target_2930,v30,fine,DrillTool\WObj:=FakeWing;
SetDO drillDone,1;
WaitUntil drillDone = 0;
        MoveL RelTool(Target_2930,0,0,-10),v30,z10,DrillTool\WObj:=FakeWing;
        MoveL RelTool(Target_2940,0,0,-10),v30,z10,DrillTool\WObj:=FakeWing;
        MoveL Target_2940,v30,fine,DrillTool\WObj:=FakeWing;
SetDO drillDone,1;
WaitUntil drillDone = 0;
        MoveL RelTool(Target_2940,0,0,-10),v30,z10,DrillTool\WObj:=FakeWing;
        MoveL RelTool(Target_2950,0,0,-10),v30,z10,DrillTool\WObj:=FakeWing;
        MoveL Target_2950,v30,fine,DrillTool\WObj:=FakeWing;
SetDO drillDone,1;
WaitUntil drillDone = 0;
        MoveL RelTool(Target_2950,0,0,-10),v30,z10,DrillTool\WObj:=FakeWing;
        MoveL RelTool(Target_2960,0,0,-10),v30,z10,DrillTool\WObj:=FakeWing;
        MoveL Target_2960,v30,fine,DrillTool\WObj:=FakeWing;
SetDO drillDone,1;
WaitUntil drillDone = 0;
        MoveL RelTool(Target_2960,0,0,-10),v30,z10,DrillTool\WObj:=FakeWing;
        MoveL RelTool(Target_2970,0,0,-10),v30,z10,DrillTool\WObj:=FakeWing;
        MoveL Target_2970,v30,fine,DrillTool\WObj:=FakeWing;
SetDO drillDone,1;
WaitUntil drillDone = 0;
        MoveL RelTool(Target_2970,0,0,-10),v30,z10,DrillTool\WObj:=FakeWing;
        MoveL RelTool(Target_2980,0,0,-10),v30,z10,DrillTool\WObj:=FakeWing;
        MoveL Target_2980,v30,fine,DrillTool\WObj:=FakeWing;
SetDO drillDone,1;
WaitUntil drillDone = 0;
        MoveL RelTool(Target_2980,0,0,-10),v30,z10,DrillTool\WObj:=FakeWing;
        MoveL RelTool(Target_2990,0,0,-10),v30,z10,DrillTool\WObj:=FakeWing;
        MoveL Target_2990,v30,fine,DrillTool\WObj:=FakeWing;
SetDO drillDone,1;
WaitUntil drillDone = 0;
        MoveL RelTool(Target_2990,0,0,-10),v30,z10,DrillTool\WObj:=FakeWing;
        MoveL RelTool(Target_3000,0,0,-10),v30,z10,DrillTool\WObj:=FakeWing;
        MoveL Target_3000,v30,fine,DrillTool\WObj:=FakeWing;
SetDO drillDone,1;
WaitUntil drillDone = 0;
        MoveL RelTool(Target_3000,0,0,-10),v30,z10,DrillTool\WObj:=FakeWing;
        MoveL RelTool(Target_3010,0,0,-10),v30,z10,DrillTool\WObj:=FakeWing;
        MoveL Target_3010,v30,fine,DrillTool\WObj:=FakeWing;
SetDO drillDone,1;
WaitUntil drillDone = 0;
        MoveL RelTool(Target_3010,0,0,-10),v30,z10,DrillTool\WObj:=FakeWing;
        MoveL RelTool(Target_3020,0,0,-10),v30,z10,DrillTool\WObj:=FakeWing;
        MoveL Target_3020,v30,fine,DrillTool\WObj:=FakeWing;
SetDO drillDone,1;
WaitUntil drillDone = 0;
        MoveL RelTool(Target_3020,0,0,-10),v30,z10,DrillTool\WObj:=FakeWing;
        MoveL RelTool(Target_3030,0,0,-10),v30,z10,DrillTool\WObj:=FakeWing;
        MoveL Target_3030,v30,fine,DrillTool\WObj:=FakeWing;
SetDO drillDone,1;
WaitUntil drillDone = 0;
        MoveL RelTool(Target_3030,0,0,-10),v30,z10,DrillTool\WObj:=FakeWing;
        MoveL RelTool(Target_3040,0,0,-10),v30,z10,DrillTool\WObj:=FakeWing;
        MoveL Target_3040,v30,fine,DrillTool\WObj:=FakeWing;
SetDO drillDone,1;
WaitUntil drillDone = 0;
        MoveL RelTool(Target_3040,0,0,-10),v30,z10,DrillTool\WObj:=FakeWing;
        MoveL RelTool(Target_3050,0,0,-10),v30,z10,DrillTool\WObj:=FakeWing;
        MoveL Target_3050,v30,fine,DrillTool\WObj:=FakeWing;
SetDO drillDone,1;
WaitUntil drillDone = 0;
        MoveL RelTool(Target_3050,0,0,-10),v30,z10,DrillTool\WObj:=FakeWing;
        MoveL RelTool(Target_3060,0,0,-10),v30,z10,DrillTool\WObj:=FakeWing;
        MoveL Target_3060,v30,fine,DrillTool\WObj:=FakeWing;
SetDO drillDone,1;
WaitUntil drillDone = 0;
        MoveL RelTool(Target_3060,0,0,-10),v30,z10,DrillTool\WObj:=FakeWing;
        MoveL RelTool(Target_3070,0,0,-10),v30,z10,DrillTool\WObj:=FakeWing;
        MoveL Target_3070,v30,fine,DrillTool\WObj:=FakeWing;
SetDO drillDone,1;
WaitUntil drillDone = 0;
        MoveL RelTool(Target_3070,0,0,-10),v30,z10,DrillTool\WObj:=FakeWing;
        MoveL RelTool(Target_3080,0,0,-10),v30,z10,DrillTool\WObj:=FakeWing;
        MoveL Target_3080,v30,fine,DrillTool\WObj:=FakeWing;
SetDO drillDone,1;
WaitUntil drillDone = 0;
        MoveL RelTool(Target_3080,0,0,-10),v30,z10,DrillTool\WObj:=FakeWing;
        MoveL RelTool(Target_3090,0,0,-10),v30,z10,DrillTool\WObj:=FakeWing;
        MoveL Target_3090,v30,fine,DrillTool\WObj:=FakeWing;
SetDO drillDone,1;
WaitUntil drillDone = 0;
        MoveL RelTool(Target_3090,0,0,-10),v30,z10,DrillTool\WObj:=FakeWing;
        MoveL RelTool(Target_3100,0,0,-10),v30,z10,DrillTool\WObj:=FakeWing;
        MoveL Target_3100,v30,fine,DrillTool\WObj:=FakeWing;
SetDO drillDone,1;
WaitUntil drillDone = 0;
        MoveL RelTool(Target_3100,0,0,-10),v30,z10,DrillTool\WObj:=FakeWing;
        MoveL RelTool(Target_3110,0,0,-10),v30,z10,DrillTool\WObj:=FakeWing;
        MoveL Target_3110,v30,fine,DrillTool\WObj:=FakeWing;
SetDO drillDone,1;
WaitUntil drillDone = 0;
        MoveL RelTool(Target_3110,0,0,-10),v30,z10,DrillTool\WObj:=FakeWing;
        MoveL RelTool(Target_3120,0,0,-10),v30,z10,DrillTool\WObj:=FakeWing;
        MoveL Target_3120,v30,fine,DrillTool\WObj:=FakeWing;
SetDO drillDone,1;
WaitUntil drillDone = 0;
        MoveL RelTool(Target_3120,0,0,-10),v30,z10,DrillTool\WObj:=FakeWing;
        MoveL RelTool(Target_3130,0,0,-10),v30,z10,DrillTool\WObj:=FakeWing;
        MoveL Target_3130,v30,fine,DrillTool\WObj:=FakeWing;
SetDO drillDone,1;
WaitUntil drillDone = 0;
        MoveL RelTool(Target_3130,0,0,-10),v30,z10,DrillTool\WObj:=FakeWing;
        MoveL RelTool(Target_3140,0,0,-10),v30,z10,DrillTool\WObj:=FakeWing;
        MoveL Target_3140,v30,fine,DrillTool\WObj:=FakeWing;
SetDO drillDone,1;
WaitUntil drillDone = 0;
        MoveL RelTool(Target_3140,0,0,-10),v30,z10,DrillTool\WObj:=FakeWing;
        MoveL RelTool(Target_3150,0,0,-10),v30,z10,DrillTool\WObj:=FakeWing;
        MoveL Target_3150,v30,fine,DrillTool\WObj:=FakeWing;
SetDO drillDone,1;
WaitUntil drillDone = 0;
        MoveL RelTool(Target_3150,0,0,-10),v30,z10,DrillTool\WObj:=FakeWing;
        MoveL RelTool(Target_3160,0,0,-10),v30,z10,DrillTool\WObj:=FakeWing;
        MoveL Target_3160,v30,fine,DrillTool\WObj:=FakeWing;
SetDO drillDone,1;
WaitUntil drillDone = 0;
        MoveL RelTool(Target_3160,0,0,-10),v30,z10,DrillTool\WObj:=FakeWing;
        MoveL RelTool(Target_3170,0,0,-10),v30,z10,DrillTool\WObj:=FakeWing;
        MoveL Target_3170,v30,fine,DrillTool\WObj:=FakeWing;
SetDO drillDone,1;
WaitUntil drillDone = 0;
        MoveL RelTool(Target_3170,0,0,-10),v30,z10,DrillTool\WObj:=FakeWing;
        MoveL RelTool(Target_3180,0,0,-10),v30,z10,DrillTool\WObj:=FakeWing;
        MoveL Target_3180,v30,fine,DrillTool\WObj:=FakeWing;
SetDO drillDone,1;
WaitUntil drillDone = 0;
        MoveL RelTool(Target_3180,0,0,-10),v30,z10,DrillTool\WObj:=FakeWing;
        MoveL RelTool(Target_3190,0,0,-10),v30,z10,DrillTool\WObj:=FakeWing;
        MoveL Target_3190,v30,fine,DrillTool\WObj:=FakeWing;
SetDO drillDone,1;
WaitUntil drillDone = 0;
        MoveL RelTool(Target_3190,0,0,-10),v30,z10,DrillTool\WObj:=FakeWing;
        MoveL RelTool(Target_3200,0,0,-10),v30,z10,DrillTool\WObj:=FakeWing;
        MoveL Target_3200,v30,fine,DrillTool\WObj:=FakeWing;
SetDO drillDone,1;
WaitUntil drillDone = 0;
        MoveL RelTool(Target_3200,0,0,-10),v30,z10,DrillTool\WObj:=FakeWing;
        MoveL RelTool(Target_3210,0,0,-10),v30,z10,DrillTool\WObj:=FakeWing;
        MoveL Target_3210,v30,fine,DrillTool\WObj:=FakeWing;
SetDO drillDone,1;
WaitUntil drillDone = 0;
        MoveL RelTool(Target_3210,0,0,-10),v30,z10,DrillTool\WObj:=FakeWing;
        MoveL RelTool(Target_3220,0,0,-10),v30,z10,DrillTool\WObj:=FakeWing;
        MoveL Target_3220,v30,fine,DrillTool\WObj:=FakeWing;
SetDO drillDone,1;
WaitUntil drillDone = 0;
        MoveL RelTool(Target_3220,0,0,-10),v30,z10,DrillTool\WObj:=FakeWing;
        MoveL RelTool(Target_3230,0,0,-10),v30,z10,DrillTool\WObj:=FakeWing;
        MoveL Target_3230,v30,fine,DrillTool\WObj:=FakeWing;
SetDO drillDone,1;
WaitUntil drillDone = 0;
        MoveL RelTool(Target_3230,0,0,-10),v30,z10,DrillTool\WObj:=FakeWing;
        MoveL RelTool(Target_3240,0,0,-10),v30,z10,DrillTool\WObj:=FakeWing;
        MoveL Target_3240,v30,fine,DrillTool\WObj:=FakeWing;
SetDO drillDone,1;
WaitUntil drillDone = 0;
        MoveL RelTool(Target_3240,0,0,-10),v30,z10,DrillTool\WObj:=FakeWing;
        MoveL RelTool(Target_3250,0,0,-10),v30,z10,DrillTool\WObj:=FakeWing;
        MoveL Target_3250,v30,fine,DrillTool\WObj:=FakeWing;
SetDO drillDone,1;
WaitUntil drillDone = 0;
        MoveL RelTool(Target_3250,0,0,-10),v30,z10,DrillTool\WObj:=FakeWing;
        MoveL RelTool(Target_3260,0,0,-10),v30,z10,DrillTool\WObj:=FakeWing;
        MoveL Target_3260,v30,fine,DrillTool\WObj:=FakeWing;
SetDO drillDone,1;
WaitUntil drillDone = 0;
        MoveL RelTool(Target_3260,0,0,-10),v30,z10,DrillTool\WObj:=FakeWing;
        MoveL RelTool(Target_3270,0,0,-10),v30,z10,DrillTool\WObj:=FakeWing;
        MoveL Target_3270,v30,fine,DrillTool\WObj:=FakeWing;
SetDO drillDone,1;
WaitUntil drillDone = 0;
        MoveL RelTool(Target_3270,0,0,-10),v30,z10,DrillTool\WObj:=FakeWing;
        MoveL RelTool(Target_3280,0,0,-10),v30,z10,DrillTool\WObj:=FakeWing;
        MoveL Target_3280,v30,fine,DrillTool\WObj:=FakeWing;
SetDO drillDone,1;
WaitUntil drillDone = 0;
        MoveL RelTool(Target_3280,0,0,-10),v30,z10,DrillTool\WObj:=FakeWing;
        MoveL RelTool(Target_3290,0,0,-10),v30,z10,DrillTool\WObj:=FakeWing;
        MoveL Target_3290,v30,fine,DrillTool\WObj:=FakeWing;
SetDO drillDone,1;
WaitUntil drillDone = 0;
        MoveL RelTool(Target_3290,0,0,-10),v30,z10,DrillTool\WObj:=FakeWing;
        MoveL RelTool(Target_3300,0,0,-10),v30,z10,DrillTool\WObj:=FakeWing;
        MoveL Target_3300,v30,fine,DrillTool\WObj:=FakeWing;
SetDO drillDone,1;
WaitUntil drillDone = 0;
        MoveL RelTool(Target_3300,0,0,-10),v30,z10,DrillTool\WObj:=FakeWing;
        MoveL RelTool(Target_3310,0,0,-10),v30,z10,DrillTool\WObj:=FakeWing;
        MoveL Target_3310,v30,fine,DrillTool\WObj:=FakeWing;
SetDO drillDone,1;
WaitUntil drillDone = 0;
        MoveL RelTool(Target_3310,0,0,-10),v30,z10,DrillTool\WObj:=FakeWing;
        MoveL RelTool(Target_3320,0,0,-10),v30,z10,DrillTool\WObj:=FakeWing;
        MoveL Target_3320,v30,fine,DrillTool\WObj:=FakeWing;
SetDO drillDone,1;
WaitUntil drillDone = 0;
        MoveL RelTool(Target_3320,0,0,-10),v30,z10,DrillTool\WObj:=FakeWing;
        MoveL RelTool(Target_3330,0,0,-10),v30,z10,DrillTool\WObj:=FakeWing;
        MoveL Target_3330,v30,fine,DrillTool\WObj:=FakeWing;
SetDO drillDone,1;
WaitUntil drillDone = 0;
        MoveL RelTool(Target_3330,0,0,-10),v30,z10,DrillTool\WObj:=FakeWing;
        MoveL RelTool(Target_3340,0,0,-10),v30,z10,DrillTool\WObj:=FakeWing;
        MoveL Target_3340,v30,fine,DrillTool\WObj:=FakeWing;
SetDO drillDone,1;
WaitUntil drillDone = 0;
        MoveL RelTool(Target_3340,0,0,-10),v30,z10,DrillTool\WObj:=FakeWing;
        MoveL RelTool(Target_3350,0,0,-10),v30,z10,DrillTool\WObj:=FakeWing;
        MoveL Target_3350,v30,fine,DrillTool\WObj:=FakeWing;
SetDO drillDone,1;
WaitUntil drillDone = 0;
        MoveL RelTool(Target_3350,0,0,-10),v30,z10,DrillTool\WObj:=FakeWing;
        MoveL RelTool(Target_3360,0,0,-10),v30,z10,DrillTool\WObj:=FakeWing;
        MoveL Target_3360,v30,fine,DrillTool\WObj:=FakeWing;
SetDO drillDone,1;
WaitUntil drillDone = 0;
        MoveL RelTool(Target_3360,0,0,-10),v30,z10,DrillTool\WObj:=FakeWing;
        MoveL RelTool(Target_3370,0,0,-10),v30,z10,DrillTool\WObj:=FakeWing;
        MoveL Target_3370,v30,fine,DrillTool\WObj:=FakeWing;
SetDO drillDone,1;
WaitUntil drillDone = 0;
        MoveL RelTool(Target_3370,0,0,-10),v30,z10,DrillTool\WObj:=FakeWing;
        MoveL RelTool(Target_3380,0,0,-10),v30,z10,DrillTool\WObj:=FakeWing;
        MoveL Target_3380,v30,fine,DrillTool\WObj:=FakeWing;
SetDO drillDone,1;
WaitUntil drillDone = 0;
        MoveL RelTool(Target_3380,0,0,-10),v30,z10,DrillTool\WObj:=FakeWing;
        MoveL RelTool(Target_3390,0,0,-10),v30,z10,DrillTool\WObj:=FakeWing;
        MoveL Target_3390,v30,fine,DrillTool\WObj:=FakeWing;
SetDO drillDone,1;
WaitUntil drillDone = 0;
        MoveL RelTool(Target_3390,0,0,-10),v30,z10,DrillTool\WObj:=FakeWing;
        MoveL RelTool(Target_3400,0,0,-10),v30,z10,DrillTool\WObj:=FakeWing;
        MoveL Target_3400,v30,fine,DrillTool\WObj:=FakeWing;
SetDO drillDone,1;
WaitUntil drillDone = 0;
        MoveL RelTool(Target_3400,0,0,-10),v30,z10,DrillTool\WObj:=FakeWing;
        MoveL RelTool(Target_3410,0,0,-10),v30,z10,DrillTool\WObj:=FakeWing;
        MoveL Target_3410,v30,fine,DrillTool\WObj:=FakeWing;
SetDO drillDone,1;
WaitUntil drillDone = 0;
        MoveL RelTool(Target_3410,0,0,-10),v30,z10,DrillTool\WObj:=FakeWing;
        MoveL RelTool(Target_3420,0,0,-10),v30,z10,DrillTool\WObj:=FakeWing;
        MoveL Target_3420,v30,fine,DrillTool\WObj:=FakeWing;
SetDO drillDone,1;
WaitUntil drillDone = 0;
        MoveL RelTool(Target_3420,0,0,-10),v30,z10,DrillTool\WObj:=FakeWing;
        MoveL RelTool(Target_3430,0,0,-10),v30,z10,DrillTool\WObj:=FakeWing;
        MoveL Target_3430,v30,fine,DrillTool\WObj:=FakeWing;
SetDO drillDone,1;
WaitUntil drillDone = 0;
        MoveL RelTool(Target_3430,0,0,-10),v30,z10,DrillTool\WObj:=FakeWing;
        MoveL RelTool(Target_3440,0,0,-10),v30,z10,DrillTool\WObj:=FakeWing;
        MoveL Target_3440,v30,fine,DrillTool\WObj:=FakeWing;
SetDO drillDone,1;
WaitUntil drillDone = 0;
        MoveL RelTool(Target_3440,0,0,-10),v30,z10,DrillTool\WObj:=FakeWing;
        MoveL RelTool(Target_3450,0,0,-10),v30,z10,DrillTool\WObj:=FakeWing;
        MoveL Target_3450,v30,fine,DrillTool\WObj:=FakeWing;
SetDO drillDone,1;
WaitUntil drillDone = 0;
        MoveL RelTool(Target_3450,0,0,-10),v30,z10,DrillTool\WObj:=FakeWing;
        MoveL RelTool(Target_3460,0,0,-10),v30,z10,DrillTool\WObj:=FakeWing;
        MoveL Target_3460,v30,fine,DrillTool\WObj:=FakeWing;
SetDO drillDone,1;
WaitUntil drillDone = 0;
        MoveL RelTool(Target_3460,0,0,-10),v30,z10,DrillTool\WObj:=FakeWing;
        MoveL RelTool(Target_3470,0,0,-10),v30,z10,DrillTool\WObj:=FakeWing;
        MoveL Target_3470,v30,fine,DrillTool\WObj:=FakeWing;
SetDO drillDone,1;
WaitUntil drillDone = 0;
        MoveL RelTool(Target_3470,0,0,-10),v30,z10,DrillTool\WObj:=FakeWing;
        MoveL RelTool(Target_3480,0,0,-10),v30,z10,DrillTool\WObj:=FakeWing;
        MoveL Target_3480,v30,fine,DrillTool\WObj:=FakeWing;
SetDO drillDone,1;
WaitUntil drillDone = 0;
        MoveL RelTool(Target_3480,0,0,-10),v30,z10,DrillTool\WObj:=FakeWing;
        MoveL RelTool(Target_3490,0,0,-10),v30,z10,DrillTool\WObj:=FakeWing;
        MoveL Target_3490,v30,fine,DrillTool\WObj:=FakeWing;
SetDO drillDone,1;
WaitUntil drillDone = 0;
        MoveL RelTool(Target_3490,0,0,-10),v30,z10,DrillTool\WObj:=FakeWing;
        MoveL RelTool(Target_3500,0,0,-10),v30,z10,DrillTool\WObj:=FakeWing;
        MoveL Target_3500,v30,fine,DrillTool\WObj:=FakeWing;
SetDO drillDone,1;
WaitUntil drillDone = 0;
        MoveL RelTool(Target_3500,0,0,-10),v30,z10,DrillTool\WObj:=FakeWing;
        MoveL RelTool(Target_3510,0,0,-10),v30,z10,DrillTool\WObj:=FakeWing;
        MoveL Target_3510,v30,fine,DrillTool\WObj:=FakeWing;
SetDO drillDone,1;
WaitUntil drillDone = 0;
        MoveL RelTool(Target_3510,0,0,-10),v30,z10,DrillTool\WObj:=FakeWing;
        MoveL RelTool(Target_3520,0,0,-10),v30,z10,DrillTool\WObj:=FakeWing;
        MoveL Target_3520,v30,fine,DrillTool\WObj:=FakeWing;
SetDO drillDone,1;
WaitUntil drillDone = 0;
        MoveL RelTool(Target_3520,0,0,-10),v30,z10,DrillTool\WObj:=FakeWing;
        MoveL RelTool(Target_3530,0,0,-10),v30,z10,DrillTool\WObj:=FakeWing;
        MoveL Target_3530,v30,fine,DrillTool\WObj:=FakeWing;
SetDO drillDone,1;
WaitUntil drillDone = 0;
        MoveL RelTool(Target_3530,0,0,-10),v30,z10,DrillTool\WObj:=FakeWing;
        MoveL RelTool(Target_3540,0,0,-10),v30,z10,DrillTool\WObj:=FakeWing;
        MoveL Target_3540,v30,fine,DrillTool\WObj:=FakeWing;
SetDO drillDone,1;
WaitUntil drillDone = 0;
        MoveL RelTool(Target_3540,0,0,-10),v30,z10,DrillTool\WObj:=FakeWing;
        MoveL RelTool(Target_3550,0,0,-10),v30,z10,DrillTool\WObj:=FakeWing;
        MoveL Target_3550,v30,fine,DrillTool\WObj:=FakeWing;
SetDO drillDone,1;
WaitUntil drillDone = 0;
        MoveL RelTool(Target_3550,0,0,-10),v30,z10,DrillTool\WObj:=FakeWing;
        MoveL RelTool(Target_3560,0,0,-10),v30,z10,DrillTool\WObj:=FakeWing;
        MoveL Target_3560,v30,fine,DrillTool\WObj:=FakeWing;
SetDO drillDone,1;
WaitUntil drillDone = 0;
        MoveL RelTool(Target_3560,0,0,-10),v30,z10,DrillTool\WObj:=FakeWing;
        MoveL RelTool(Target_3570,0,0,-10),v30,z10,DrillTool\WObj:=FakeWing;
        MoveL Target_3570,v30,fine,DrillTool\WObj:=FakeWing;
SetDO drillDone,1;
WaitUntil drillDone = 0;
        MoveL RelTool(Target_3570,0,0,-10),v30,z10,DrillTool\WObj:=FakeWing;
        MoveL RelTool(Target_3580,0,0,-10),v30,z10,DrillTool\WObj:=FakeWing;
        MoveL Target_3580,v30,fine,DrillTool\WObj:=FakeWing;
SetDO drillDone,1;
WaitUntil drillDone = 0;
        MoveL RelTool(Target_3580,0,0,-10),v30,z10,DrillTool\WObj:=FakeWing;
        MoveL RelTool(Target_3590,0,0,-10),v30,z10,DrillTool\WObj:=FakeWing;
        MoveL Target_3590,v30,fine,DrillTool\WObj:=FakeWing;
SetDO drillDone,1;
WaitUntil drillDone = 0;
        MoveL RelTool(Target_3590,0,0,-10),v30,z10,DrillTool\WObj:=FakeWing;
        MoveL RelTool(Target_3600,0,0,-10),v30,z10,DrillTool\WObj:=FakeWing;
        MoveL Target_3600,v30,fine,DrillTool\WObj:=FakeWing;
SetDO drillDone,1;
WaitUntil drillDone = 0;
        MoveL RelTool(Target_3600,0,0,-10),v30,z10,DrillTool\WObj:=FakeWing;
        MoveL RelTool(Target_3610,0,0,-10),v30,z10,DrillTool\WObj:=FakeWing;
        MoveL Target_3610,v30,fine,DrillTool\WObj:=FakeWing;
SetDO drillDone,1;
WaitUntil drillDone = 0;
        MoveL RelTool(Target_3610,0,0,-10),v30,z10,DrillTool\WObj:=FakeWing;
        MoveL RelTool(Target_3620,0,0,-10),v30,z10,DrillTool\WObj:=FakeWing;
        MoveL Target_3620,v30,fine,DrillTool\WObj:=FakeWing;
SetDO drillDone,1;
WaitUntil drillDone = 0;
        MoveL RelTool(Target_3620,0,0,-10),v30,z10,DrillTool\WObj:=FakeWing;
        MoveL RelTool(Target_3630,0,0,-10),v30,z10,DrillTool\WObj:=FakeWing;
        MoveL Target_3630,v30,fine,DrillTool\WObj:=FakeWing;
SetDO drillDone,1;
WaitUntil drillDone = 0;
        MoveL RelTool(Target_3630,0,0,-10),v30,z10,DrillTool\WObj:=FakeWing;
        MoveL RelTool(Target_3640,0,0,-10),v30,z10,DrillTool\WObj:=FakeWing;
        MoveL Target_3640,v30,fine,DrillTool\WObj:=FakeWing;
SetDO drillDone,1;
WaitUntil drillDone = 0;
        MoveL RelTool(Target_3640,0,0,-10),v30,z10,DrillTool\WObj:=FakeWing;
        MoveL RelTool(Target_3650,0,0,-10),v30,z10,DrillTool\WObj:=FakeWing;
        MoveL Target_3650,v30,fine,DrillTool\WObj:=FakeWing;
SetDO drillDone,1;
WaitUntil drillDone = 0;
        MoveL RelTool(Target_3650,0,0,-10),v30,z10,DrillTool\WObj:=FakeWing;
        MoveL RelTool(Target_3660,0,0,-10),v30,z10,DrillTool\WObj:=FakeWing;
        MoveL Target_3660,v30,fine,DrillTool\WObj:=FakeWing;
SetDO drillDone,1;
WaitUntil drillDone = 0;
        MoveL RelTool(Target_3660,0,0,-10),v30,z10,DrillTool\WObj:=FakeWing;
        MoveL RelTool(Target_3670,0,0,-10),v30,z10,DrillTool\WObj:=FakeWing;
        MoveL Target_3670,v30,fine,DrillTool\WObj:=FakeWing;
SetDO drillDone,1;
WaitUntil drillDone = 0;
        MoveL RelTool(Target_3670,0,0,-10),v30,z10,DrillTool\WObj:=FakeWing;
        MoveL RelTool(Target_3680,0,0,-10),v30,z10,DrillTool\WObj:=FakeWing;
        MoveL Target_3680,v30,fine,DrillTool\WObj:=FakeWing;
SetDO drillDone,1;
WaitUntil drillDone = 0;
        MoveL RelTool(Target_3680,0,0,-10),v30,z10,DrillTool\WObj:=FakeWing;
        MoveL RelTool(Target_3690,0,0,-10),v30,z10,DrillTool\WObj:=FakeWing;
        MoveL Target_3690,v30,fine,DrillTool\WObj:=FakeWing;
SetDO drillDone,1;
WaitUntil drillDone = 0;
        MoveL RelTool(Target_3690,0,0,-10),v30,z10,DrillTool\WObj:=FakeWing;
        MoveL RelTool(Target_3700,0,0,-10),v30,z10,DrillTool\WObj:=FakeWing;
        MoveL Target_3700,v30,fine,DrillTool\WObj:=FakeWing;
SetDO drillDone,1;
WaitUntil drillDone = 0;
        MoveL RelTool(Target_3700,0,0,-10),v30,z10,DrillTool\WObj:=FakeWing;
        MoveL RelTool(Target_3710,0,0,-10),v30,z10,DrillTool\WObj:=FakeWing;
        MoveL Target_3710,v30,fine,DrillTool\WObj:=FakeWing;
SetDO drillDone,1;
WaitUntil drillDone = 0;
        MoveL RelTool(Target_3710,0,0,-10),v30,z10,DrillTool\WObj:=FakeWing;
        MoveL RelTool(Target_3720,0,0,-10),v30,z10,DrillTool\WObj:=FakeWing;
        MoveL Target_3720,v30,fine,DrillTool\WObj:=FakeWing;
SetDO drillDone,1;
WaitUntil drillDone = 0;
        MoveL RelTool(Target_3720,0,0,-10),v30,z10,DrillTool\WObj:=FakeWing;
        MoveL RelTool(Target_3730,0,0,-10),v30,z10,DrillTool\WObj:=FakeWing;
        MoveL Target_3730,v30,fine,DrillTool\WObj:=FakeWing;
SetDO drillDone,1;
WaitUntil drillDone = 0;
        MoveL RelTool(Target_3730,0,0,-10),v30,z10,DrillTool\WObj:=FakeWing;
        MoveL RelTool(Target_3740,0,0,-10),v30,z10,DrillTool\WObj:=FakeWing;
        MoveL Target_3740,v30,fine,DrillTool\WObj:=FakeWing;
SetDO drillDone,1;
WaitUntil drillDone = 0;
        MoveL RelTool(Target_3740,0,0,-10),v30,z10,DrillTool\WObj:=FakeWing;
        MoveL RelTool(Target_3750,0,0,-10),v30,z10,DrillTool\WObj:=FakeWing;
        MoveL Target_3750,v30,fine,DrillTool\WObj:=FakeWing;
SetDO drillDone,1;
WaitUntil drillDone = 0;
        MoveL RelTool(Target_3750,0,0,-10),v30,z10,DrillTool\WObj:=FakeWing;
        MoveL RelTool(Target_3760,0,0,-10),v30,z10,DrillTool\WObj:=FakeWing;
        MoveL Target_3760,v30,fine,DrillTool\WObj:=FakeWing;
SetDO drillDone,1;
WaitUntil drillDone = 0;
        MoveL RelTool(Target_3760,0,0,-10),v30,z10,DrillTool\WObj:=FakeWing;
        MoveL RelTool(Target_3770,0,0,-10),v30,z10,DrillTool\WObj:=FakeWing;
        MoveL Target_3770,v30,fine,DrillTool\WObj:=FakeWing;
SetDO drillDone,1;
WaitUntil drillDone = 0;
        MoveL RelTool(Target_3770,0,0,-10),v30,z10,DrillTool\WObj:=FakeWing;
        MoveL RelTool(Target_3780,0,0,-10),v30,z10,DrillTool\WObj:=FakeWing;
        MoveL Target_3780,v30,fine,DrillTool\WObj:=FakeWing;
SetDO drillDone,1;
WaitUntil drillDone = 0;
        MoveL RelTool(Target_3780,0,0,-10),v30,z10,DrillTool\WObj:=FakeWing;
        MoveL RelTool(Target_3790,0,0,-10),v30,z10,DrillTool\WObj:=FakeWing;
        MoveL Target_3790,v30,fine,DrillTool\WObj:=FakeWing;
SetDO drillDone,1;
WaitUntil drillDone = 0;
        MoveL RelTool(Target_3790,0,0,-10),v30,z10,DrillTool\WObj:=FakeWing;
        MoveL RelTool(Target_3800,0,0,-10),v30,z10,DrillTool\WObj:=FakeWing;
        MoveL Target_3800,v30,fine,DrillTool\WObj:=FakeWing;
SetDO drillDone,1;
WaitUntil drillDone = 0;
        MoveL RelTool(Target_3800,0,0,-10),v30,z10,DrillTool\WObj:=FakeWing;
        MoveL RelTool(Target_3810,0,0,-10),v30,z10,DrillTool\WObj:=FakeWing;
        MoveL Target_3810,v30,fine,DrillTool\WObj:=FakeWing;
SetDO drillDone,1;
WaitUntil drillDone = 0;
        MoveL RelTool(Target_3810,0,0,-10),v30,z10,DrillTool\WObj:=FakeWing;
        MoveL RelTool(Target_3820,0,0,-10),v30,z10,DrillTool\WObj:=FakeWing;
        MoveL Target_3820,v30,fine,DrillTool\WObj:=FakeWing;
SetDO drillDone,1;
WaitUntil drillDone = 0;
        MoveL RelTool(Target_3820,0,0,-10),v30,z10,DrillTool\WObj:=FakeWing;
        MoveL RelTool(Target_3830,0,0,-10),v30,z10,DrillTool\WObj:=FakeWing;
        MoveL Target_3830,v30,fine,DrillTool\WObj:=FakeWing;
SetDO drillDone,1;
WaitUntil drillDone = 0;
        MoveL RelTool(Target_3830,0,0,-10),v30,z10,DrillTool\WObj:=FakeWing;
        MoveL RelTool(Target_3840,0,0,-10),v30,z10,DrillTool\WObj:=FakeWing;
        MoveL Target_3840,v30,fine,DrillTool\WObj:=FakeWing;
SetDO drillDone,1;
WaitUntil drillDone = 0;
        MoveL RelTool(Target_3840,0,0,-10),v30,z10,DrillTool\WObj:=FakeWing;
        MoveL RelTool(Target_3850,0,0,-10),v30,z10,DrillTool\WObj:=FakeWing;
        MoveL Target_3850,v30,fine,DrillTool\WObj:=FakeWing;
SetDO drillDone,1;
WaitUntil drillDone = 0;
        MoveL RelTool(Target_3850,0,0,-10),v30,z10,DrillTool\WObj:=FakeWing;
        MoveL RelTool(Target_3860,0,0,-10),v30,z10,DrillTool\WObj:=FakeWing;
        MoveL Target_3860,v30,fine,DrillTool\WObj:=FakeWing;
